METHOD FINAL metMbSerialClient
VAR_IN_OUT
	tTimeOut	: TIME;
	utQuery	    : WagoAppPlcModbus.typMbQuery;
	xTrigger	: BOOL;
	utResponse	: WagoAppPlcModbus.typMbResponse;
END_VAR
VAR_OUTPUT
	xError	: BOOL;
	uiID	: UINT;
END_VAR
VAR
	xDumyTrigger	:	BOOL;
END_VAR
IF NOT fbConfigFile.xError THEN
	(* Clear Call on Error*)
	IF fbMbClientSerial.xError THEN
		fbMbClientSerial(xConnect 	:= FALSE,
						 xTrigger 	:= xDumyTrigger,
						 utQuery  	:= utQuery,
						 utResponse := utResponse);
	END_IF;				 
    fbMbClientSerial           (xConnect    := xTrigger,
                                I_Port      := I_Port,
                                udiBaudrate := scParameter.fbudiBaudrate.udiValue,
                                usiDataBits := scParameter.fbusiDataBits.usiValue,
                                eParity     := scParameter.fbiParity.iValue,
                                eStopBits   := scParameter.fbiStopBits.iValue,
                                eHandshake  := scParameter.fbiHandshake.iValue,
                                ePhysical   := scParameter.fbiPhysikal.iValue,
                                eFrameType  := SEL(scParameter.fbxRtuOrAscii.xValue,WagoAppPlcModbus.eMbFrameType.RTU,WagoAppPlcModbus.eMbFrameType.ASCII),
                                tTimeOut    := tTimeOut,
                                utQuery     := utQuery,
                                xTrigger    := xTrigger,
                                utResponse  := utResponse,
                                xError      => xError);    
								(* Status *)
                                uiID        := fbMbClientSerial.oStatus.uiID;								
ELSE
    xError := TRUE;
END_IF;
END_METHOD

ACTION actConfig:
(* Config File *)
fbConfigFile();

scParameter.fbudiBaudrate         (_usiParaNr :=  1, ItfConfigFb := fbConfigFile , _MinInit := 9600     , _MaxInit :=  115200 );
scParameter.fbusiDataBits         (_usiParaNr :=  2, ItfConfigFb := fbConfigFile , _MinInit :=    5     , _MaxInit :=       8 );
scParameter.fbiParity             (_usiParaNr :=  3, ItfConfigFb := fbConfigFile , _MinInit :=    0     , _MaxInit :=       5 );
scParameter.fbiStopBits           (_usiParaNr :=  4, ItfConfigFb := fbConfigFile , _MinInit :=    0     , _MaxInit :=       5 );
scParameter.fbiHandshake          (_usiParaNr :=  5, ItfConfigFb := fbConfigFile , _MinInit :=    0     , _MaxInit :=       7 );
scParameter.fbiPhysikal           (_usiParaNr :=  6, ItfConfigFb := fbConfigFile , _MinInit :=    0     , _MaxInit :=       6 );
scParameter.fbxRtuOrAscii         (_usiParaNr :=  7, ItfConfigFb := fbConfigFile                                              );
END_ACTION

END_FUNCTION_BLOCK

// 30 Program Organization Units/SERVER/fbModBusServer
{warning 'Each Modbus server needs 400000 bytes of dynamic memory'}
FUNCTION_BLOCK fbModBusServer IMPLEMENTS ITF_SERVER
VAR_INPUT
    I_SerialPort                    :   WagoTypesCom.I_WagoSysComBase;
END_VAR
VAR_OUTPUT
    xError                          :   BOOL;
END_VAR
VAR
    (* Memory *)
    ayxCoil                         :   POINTER TO ARRAY[0..16#FFFF] OF BOOL;
    ayxDiscretInput                 :   POINTER TO ARRAY[0..16#FFFF] OF BOOL;  
    aywInputRegister                :   POINTER TO ARRAY[0..16#FFFF] OF WORD;
    aywHoldingRegister              :   POINTER TO ARRAY[0..16#FFFF] OF WORD; 
    xMemoryError                    :   BOOL;
    xMemoryAllocate                 :   BOOL    := TRUE;
    (* Tcp *)
    fbMbServerModelTcp              :   WagoAppPlcModbus.FbMbSlaveDataModel;
    fbMbShowAccesTcp                :   WagoAppPlcModbus.FbShowMbAccessInfo;
    fbMbTcpServer                   :   WagoAppPlcModbus.FbMbServerTcp;
    scKeepAlive                     :   WagoAppPlcModbus.typKeepAlive;
    ltLastAccesTcp                  :   LTIME;
    fbLastAccesTcp                  :   CtaAppTime.fbTimeMeasurement;
    xErrorWatchDogTcp               :   BOOL;
    xErrorTcp                       :   BOOL;
    
    (* Udp *)
    fbMbServerModelUdp              :   WagoAppPlcModbus.FbMbSlaveDataModel;
    fbMbShowAccesUdp                :   WagoAppPlcModbus.FbShowMbAccessInfo;
    fbMbUdpServer                   :   WagoAppPlcModbus.fbMbServerUdp;
    ltLastAccesUdp                  :   LTIME;
    fbLastAccesUdp                  :   CtaAppTime.fbTimeMeasurement;  
    xErrorWatchDogUdp               :   BOOL;  
    xErrorUdp                       :   BOOL;
    
    (* Serial *)
    fbMbServerModelSerial           :   WagoAppPlcModbus.FbMbSlaveDataModel;
    fbMbShowAccesSerial             :   WagoAppPlcModbus.FbShowMbAccessInfo;
    fbMbRtuSerialServer             :   WagoAppPlcModbus.FbMbServerSerial;
    ltLastAccesSerial               :   LTIME;
    fbLastAccesSerial               :   CtaAppTime.fbTimeMeasurement;
    xErrorWatchDogSerial            :   BOOL;    
    xErrorSerial                    :   BOOL;
    
    (* Parameter *)
    fbConfigFile                    :   CtaSysConfig.fbConfigFile;
    scParameter                     :   scModBusServerParameter;
END_VAR

actConfig();
IF xMemoryAllocate AND NOT xMemoryError THEN
    ayxCoil             := __NEW(BOOL,16#10000);
    ayxDiscretInput     := __NEW(BOOL,16#10000);
    aywInputRegister    := __NEW(WORD,16#10000);
    aywHoldingRegister  := __NEW(WORD,16#10000);
    IF ayxCoil <> 0 AND ayxDiscretInput <> 0 AND aywInputRegister <> 0 AND aywHoldingRegister <> 0 THEN
        xMemoryAllocate     := FALSE;     
    ELSE 
        xMemoryError := TRUE;   
    END_IF;
END_IF;
IF  NOT xMemoryAllocate AND NOT xMemoryError THEN
    IF SIZEOF(ayxCoil^) = 65536 AND SIZEOF(ayxDiscretInput^) = 65536 AND SIZEOF(aywInputRegister^) = 131072 AND SIZEOF(aywHoldingRegister^) = 131072 THEN
        IF NOT fbConfigFile.xError THEN
            actModBusServerSerial();
            actModBusServerTcp();
            actModBusServerUdp();
        END_IF;    
        xMemoryError := FALSE;
    ELSE
        xMemoryError := TRUE;    
    END_IF
END_IF;
(* Error *)
xError := fbConfigFile.xError OR xErrorTcp OR xErrorUdp OR xErrorSerial OR xMemoryError;

ACTION actConfig:
(* Config File *)
fbConfigFile();

scParameter.scSerial.fbbyUnitId            (_usiParaNr :=  1, ItfConfigFb := fbConfigFile , _MinInit :=    0     , _MaxInit :=     247 ); 
scParameter.scSerial.fbxEnable             (_usiParaNr :=  2, ItfConfigFb := fbConfigFile                                              );
scParameter.scSerial.fbudiBaudrate         (_usiParaNr :=  3, ItfConfigFb := fbConfigFile , _MinInit := 9600     , _MaxInit :=   19600 );
scParameter.scSerial.fbusiDataBits         (_usiParaNr :=  4, ItfConfigFb := fbConfigFile , _MinInit :=    5     , _MaxInit :=       8 );
scParameter.scSerial.fbiParity             (_usiParaNr :=  5, ItfConfigFb := fbConfigFile , _MinInit :=    0     , _MaxInit :=       5 );
scParameter.scSerial.fbiStopBits           (_usiParaNr :=  6, ItfConfigFb := fbConfigFile , _MinInit :=    0     , _MaxInit :=       5 );
scParameter.scSerial.fbiHandshake          (_usiParaNr :=  7, ItfConfigFb := fbConfigFile , _MinInit :=    0     , _MaxInit :=       7 );
scParameter.scSerial.fbiPhysikal           (_usiParaNr :=  8, ItfConfigFb := fbConfigFile , _MinInit :=    0     , _MaxInit :=       6 );
scParameter.scSerial.fbxRtuOrAscii         (_usiParaNr :=  9, ItfConfigFb := fbConfigFile                                              );
scParameter.scSerial.fbxEnableWatchDog     (_usiParaNr := 10, ItfConfigFb := fbConfigFile                                              );
scParameter.scSerial.fbtWatchDog           (_usiParaNr := 11, ItfConfigFb := fbConfigFile , _MinInit := T#1S     , _MaxInit :=   T#10M );
scParameter.scTcp.fbxEnable                (_usiParaNr := 12, ItfConfigFb := fbConfigFile                                              );
scParameter.scTcp.fbbyUnitId               (_usiParaNr := 13, ItfConfigFb := fbConfigFile , _MinInit :=    0     , _MaxInit :=     255 ); 
scParameter.scTcp.fbwPort                  (_usiParaNr := 14, ItfConfigFb := fbConfigFile , _MinInit :=    0     , _MaxInit := 16#FFFF );
scParameter.scTcp.fbxKeepAlive             (_usiParaNr := 15, ItfConfigFb := fbConfigFile                                              );
scParameter.scTcp.fbtMaxIdleTime           (_usiParaNr := 16, ItfConfigFb := fbConfigFile , _MinInit := T#1S     , _MaxInit :=   T#10M );
scParameter.scTcp.fbtIntervall             (_usiParaNr := 17, ItfConfigFb := fbConfigFile , _MinInit := T#1S     , _MaxInit :=   T#10M );
scParameter.scTcp.fbudiProbes              (_usiParaNr := 18, ItfConfigFb := fbConfigFile , _MinInit :=    0     , _MaxInit :=     500 );
scParameter.scTcp.fbxEnableWatchDog        (_usiParaNr := 19, ItfConfigFb := fbConfigFile                                              );
scParameter.scTcp.fbtWatchDog              (_usiParaNr := 20, ItfConfigFb := fbConfigFile , _MinInit := T#50MS   , _MaxInit :=   T#10M );
scParameter.scUdp.fbxEnable                (_usiParaNr := 21, ItfConfigFb := fbConfigFile                                              );
scParameter.scUdp.fbbyUnitId               (_usiParaNr := 22, ItfConfigFb := fbConfigFile , _MinInit :=    0     , _MaxInit :=     255 ); 
scParameter.scUdp.fbwPort                  (_usiParaNr := 23, ItfConfigFb := fbConfigFile , _MinInit :=    0     , _MaxInit := 16#FFFF );
scParameter.scUdp.fbxEnableWatchDog        (_usiParaNr := 24, ItfConfigFb := fbConfigFile                                              );
scParameter.scUdp.fbtWatchDog              (_usiParaNr := 25, ItfConfigFb := fbConfigFile , _MinInit := T#1S     , _MaxInit :=   T#10M );
END_ACTION

ACTION actModBusServerTcp:
(* Server Memory Tcp*)
fbMbServerModelTcp(     bUnitId             := scParameter.scTcp.fbbyUnitId.byValue,
                        IIdentifyObject     := GVL_CtaModBus.fbDeviceName,
                        axDiscreteInputs    := ayxDiscretInput^,
                        axCoils             := ayxCoil^,
                        awInputRegisters    := aywInputRegister^,
                        awHoldingRegisters  := aywHoldingRegister^); 
                        
(* Tcp Server *)
IF scParameter.scTcp.fbxEnable.xValue THEN
    scKeepAlive.xEnable                     := scParameter.scTcp.fbxKeepAlive.xValue;
    scKeepAlive.tMaxIdleTime                := scParameter.scTcp.fbtMaxIdleTime.tValue;
    scKeepAlive.tInterval                   := scParameter.scTcp.fbtIntervall.tValue;
    scKeepAlive.udiProbes                   := scParameter.scTcp.fbudiProbes.udiValue;
    fbMbTcpServer(      xOpen               := scParameter.scTcp.fbxEnable.xValue,
                        wPort               := scParameter.scTcp.fbwPort.wValue,
                        utKeepAlive         := scKeepAlive,
                        eFrameType          := WagoAppPlcModbus.eMbFrameType.ETHERNET,
                        I_MbDataModel       := fbMbServerModelTcp.I_MbDataModel);
ELSIF fbMbTcpServer.xOpen THEN
    fbMbTcpServer(      xOpen               := FALSE,
                        I_MbDataModel       := fbMbServerModelTcp.I_MbDataModel);                           
END_IF;                        

(* Acces Info *)
fbMbShowAccesTcp    (   oMbAccessInfo := fbMbServerModelTcp.oMbAccessInfo);   

(* Acces Time *)
IF fbMbServerModelTcp.isReadAccess OR fbMbServerModelTcp.isWriteAccess THEN
    fbLastAccesTcp.Start();
    ltLastAccesTcp := fbLastAccesTcp.Stop();
ELSE
    ltLastAccesTcp := fbLastAccesTcp.Stop();
END_IF;

(* WatchDog *)
IF scParameter.scTcp.fbxEnableWatchDog.xValue THEN
    xErrorWatchDogTcp := TO_LTIME(scParameter.scTcp.fbtWatchDog.tValue) < ltLastAccesTcp;
ELSE
    xErrorWatchDogTcp := FALSE;
END_IF;

(* Error *)
xErrorTcp := fbConfigFile.xError OR fbMbServerModelTcp.xError OR fbMbTcpServer.xError OR xErrorWatchDogTcp;
END_ACTION

ACTION actModBusServerUdp:
(* Server Memory Udp*)
fbMbServerModelUdp(     bUnitId             := scParameter.scUdp.fbbyUnitId.byValue,
                        IIdentifyObject     := GVL_CtaModBus.fbDeviceName,
                        axDiscreteInputs    := ayxDiscretInput^,
                        axCoils             := ayxCoil^,
                        awInputRegisters    := aywInputRegister^,
                        awHoldingRegisters  := aywHoldingRegister^);  
                        
(* UDP Server *)
IF scParameter.scUdp.fbxEnable.xValue THEN
    fbMbUdpServer(      xOpen               := scParameter.scUdp.fbxEnable.xValue,
                        wPort               := scParameter.scUdp.fbwPort.wValue,
                        eFrameType          := WagoAppPlcModbus.eMbFrameType.ETHERNET,
                        I_MbDataModel       := fbMbServerModelUdp.I_MbDataModel);
ELSIF fbMbUdpServer.xOpen THEN
    fbMbUdpServer(      xOpen               := FALSE,
                        I_MbDataModel       := fbMbServerModelUdp.I_MbDataModel);                        
END_IF;                          

(* Acces Info *)
fbMbShowAccesUdp    (   oMbAccessInfo := fbMbServerModelUdp.oMbAccessInfo); 

(* Acces Time *)
IF fbMbServerModelUdp.isReadAccess OR fbMbServerModelUdp.isWriteAccess THEN
    fbLastAccesUdp.Start();
    ltLastAccesUdp := fbLastAccesSerial.Stop();
ELSE
    ltLastAccesUdp := fbLastAccesSerial.Stop();
END_IF;

(* WatchDog *)
IF scParameter.scUdp.fbxEnableWatchDog.xValue THEN
    xErrorWatchDogUdp := TO_LTIME(scParameter.scUdp.fbtWatchDog.tValue) < ltLastAccesUdp;
ELSE
    xErrorWatchDogUdp := FALSE;
END_IF;

(* Error *)
xErrorUdp := fbConfigFile.xError OR fbMbServerModelUdp.xError OR fbMbUdpServer.xError OR xErrorWatchDogUdp;
END_ACTION

ACTION actModBusServerSerial:
(* Server Memory Serial*)
fbMbServerModelSerial(  bUnitId             := scParameter.scSerial.fbbyUnitId.byValue,
                        IIdentifyObject     := GVL_CtaModBus.fbDeviceName,
                        axDiscreteInputs    := ayxDiscretInput^,
                        axCoils             := ayxCoil^,
                        awInputRegisters    := aywInputRegister^,
                        awHoldingRegisters  := aywHoldingRegister^);  
                        
(* SERIAL Server *)           
IF scParameter.scSerial.fbxEnable.xValue THEN    
	IF __QUERYINTERFACE(I_SerialPort,I_SerialPort) THEN
		(* Server Run*) 
		fbMbRtuSerialServer(xConnect            := scParameter.scSerial.fbxEnable.xValue,
							I_Port              := I_SerialPort,
							udiBaudrate         := scParameter.scSerial.fbudiBaudrate.udiValue,
							usiDataBits         := scParameter.scSerial.fbusiDataBits.usiValue,
							eParity             := scParameter.scSerial.fbiParity.iValue,
							eStopBits           := scParameter.scSerial.fbiStopBits.iValue,
							eHandshake          := scParameter.scSerial.fbiHandshake.iValue,
							ePhysical           := scParameter.scSerial.fbiPhysikal.iValue,
							eFrameType          := SEL(scParameter.scSerial.fbxRtuOrAscii.xValue,WagoAppPlcModbus.eMbFrameType.RTU,WagoAppPlcModbus.eMbFrameType.ASCII),
							I_MbDataModel       := fbMbServerModelSerial.I_MbDataModel);
   	END_IF;                     
    (* Acces Info *)
    fbMbShowAccesSerial (   oMbAccessInfo := fbMbServerModelSerial.oMbAccessInfo); 
    
    (* Acces Time *)
    IF fbMbServerModelSerial.isReadAccess OR fbMbServerModelSerial.isWriteAccess THEN
        fbLastAccesSerial.Start();
        ltLastAccesSerial := fbLastAccesSerial.Stop();
    ELSE
        ltLastAccesSerial := fbLastAccesSerial.Stop();
    END_IF;
    
    (* WatchDog *)
    IF scParameter.scSerial.fbxEnableWatchDog.xValue THEN
        xErrorWatchDogSerial := TO_LTIME(scParameter.scSerial.fbtWatchDog.tValue) < ltLastAccesSerial;
    ELSE
        xErrorWatchDogSerial := FALSE;
    END_IF;                        
                        
ELSIF fbMbRtuSerialServer.xConnect THEN
    (* Server Disconnect *)
    fbMbRtuSerialServer(xConnect            := FALSE,
                        I_Port              := I_SerialPort,
                        I_MbDataModel       := fbMbServerModelSerial.I_MbDataModel);   
ELSE
    xErrorWatchDogSerial := FALSE;
    ltLastAccesSerial    := fbLastAccesSerial.Stop();
END_IF;                        



(* Error *)
xErrorSerial := fbConfigFile.xError OR fbMbServerModelSerial.xError OR fbMbRtuSerialServer.xError OR xErrorWatchDogSerial;
END_ACTION

METHOD metGetCoil : BOOL
VAR_INPUT
    wAdr          : WORD;
END_VAR
IF NOT xMemoryAllocate AND NOT xMemoryError THEN
	IF wAdr >= LOWER_BOUND(ayxCoil^,1) AND wAdr <= UPPER_BOUND(ayxCoil^,1) THEN
    	metGetCoil := ayxCoil^[wAdr];
	END_IF;
END_IF;
END_METHOD

METHOD metSetDiscretInput : BOOL
VAR_INPUT
    wAdr          : WORD;
    xValue        : BOOL;
END_VAR
IF NOT xMemoryAllocate AND NOT xMemoryError THEN
	IF wAdr >= LOWER_BOUND(ayxDiscretInput^,1) AND wAdr <= UPPER_BOUND(ayxDiscretInput^,1) THEN
    	ayxDiscretInput^[wAdr] := xValue;
	END_IF;
END_IF;
END_METHOD

METHOD metGetHoldingRegister : WORD
VAR_INPUT
    wAdr          : WORD;
END_VAR
IF NOT xMemoryAllocate AND NOT xMemoryError THEN
	IF wAdr >= LOWER_BOUND(aywHoldingRegister^,1) AND wAdr <= UPPER_BOUND(aywHoldingRegister^,1) THEN
    	metGetHoldingRegister := aywHoldingRegister^[wAdr];
	END_IF;
END_IF;
END_METHOD

METHOD metSetInputRegister : BOOL
VAR_INPUT
    wAdr          : WORD;
    wValue        : WORD;
END_VAR
IF NOT xMemoryAllocate AND NOT xMemoryError THEN
	IF wAdr >= LOWER_BOUND(aywInputRegister^,1) AND wAdr <= UPPER_BOUND(aywInputRegister^,1) THEN
    	aywInputRegister^[wAdr] := wValue;
	END_IF;
END_IF;
END_METHOD

METHOD metAddSerialControll : BOOL
VAR_INPUT
    I_DataAccesListener :   WagoAppPlcModbus.I_DataAccessListener;
END_VAR
fbMbServerModelSerial.RegisterDataAccessListener(I_DataAccesListener);
END_METHOD

METHOD metAddTcpControll : BOOL
VAR_INPUT
    I_DataAccesListener :   WagoAppPlcModbus.I_DataAccessListener;
END_VAR
fbMbServerModelTcp.RegisterDataAccessListener(I_DataAccesListener);
END_METHOD

METHOD metAddUdpControll : BOOL
VAR_INPUT
    I_DataAccesListener :   WagoAppPlcModbus.I_DataAccessListener;
END_VAR
fbMbServerModelUdp.RegisterDataAccessListener(I_DataAccesListener);
END_METHOD

METHOD metSetHoldingRegister : BOOL
VAR_INPUT
    wAdr          : WORD;
    wValue        : WORD;
END_VAR
IF NOT xMemoryAllocate AND NOT xMemoryError THEN
	IF wAdr >= LOWER_BOUND(aywHoldingRegister^,1) AND wAdr <= UPPER_BOUND(aywHoldingRegister^,1) THEN
    	aywHoldingRegister^[wAdr] := wValue;
	END_IF;
END_IF;
END_METHOD

METHOD metSetCoil : BOOL
VAR_INPUT
    wAdr          : WORD;
    xValue        : BOOL;
END_VAR
IF NOT xMemoryAllocate AND NOT xMemoryError THEN
	IF wAdr >= LOWER_BOUND(ayxCoil^,1) AND wAdr <= UPPER_BOUND(ayxCoil^,1) THEN
    	ayxCoil^[wAdr] := xValue;
	END_IF;
END_IF;
END_METHOD

END_FUNCTION_BLOCK

// 21 Interface/SERVER/ITF_SERVER
INTERFACE ITF_SERVER EXTENDS CtaAppModbus.ITF_SERVER

METHOD metAddSerialControll : BOOL
VAR_INPUT
    I_DataAccesListener :   WagoAppPlcModbus.I_DataAccessListener;
END_VAR
END_METHOD

METHOD metAddTcpControll : BOOL
VAR_INPUT
    I_DataAccesListener :   WagoAppPlcModbus.I_DataAccessListener;
END_VAR
END_METHOD

METHOD metAddUdpControll : BOOL
VAR_INPUT
    I_DataAccesListener :   WagoAppPlcModbus.I_DataAccessListener;
END_VAR
END_METHOD

END_INTERFACE

// 30 Program Organization Units/CLIENT/NETWORK Client/TCP/fbMbTcpClient
FUNCTION_BLOCK fbMbTcpClient EXTENDS CtaSysBase.fbBASE IMPLEMENTS ITF_MbClient ,ITF_TCP_NODE                 
VAR_INPUT
    ITF_MbPortControll          : ITF_MbPortControllTcp;   
END_VAR
VAR_OUTPUT                      
    xError                      : BOOL;
END_VAR
VAR    
    (* Tcp Client *)
	ITF_BMK 					: CtaAppBmk.ITF_BMK;			
    xComAktive                  : BOOL;
    xDisabled                   : BOOL;
    xAllJobsDone                : BOOL;
    bIdOfCall                   : BYTE;
    byUnitId                    : BYTE;
    ITF_MbPortControllQuerry    : ITF_MbPortControllTcp;
    xPortControllError          : BOOL;
    scKeepAlive                 : WagoAppPlcModbus.typKeepAlive;
    xErrorMbClientTcp           : BOOL;
    uiIdMbClientTcp             : UINT;

    (* Main State *)
    uiCountErrors               : UINT;   
    usiState                    : USINT := 1;
    fbTIMEFcs                   : CtaAppTime.fbTimeMeasurement;
    ltMessungFcs                : LTIME; 
    
    (* Scan Rate *)
    TON_ScanRate                : TON;
    tonDelayRead				: Standard.TON;
	tonDelayWrite				: Standard.TON;
	xTrigDelayRead				: BOOL;
	xTrigDelayWrite				: BOOL;        
    (* FC1 *)
    fbJobFc1                    : fbJOB;
    xTrigFc1                    : BOOL;
    fbTIMEFc1                   : CtaAppTime.fbTimeMeasurement;
    ltMessungFc1                : LTIME;   
    (* FC2 *)
    fbJobFc2                    : fbJOB;
    xTrigFc2                    : BOOL; 
    fbTIMEFc2                   : CtaAppTime.fbTimeMeasurement;
    ltMessungFc2                : LTIME;    
    (* FC3 *)
    fbJobFc3                    : fbJOB;
    xTrigFc3                    : BOOL;      
    fbTIMEFc3                   : CtaAppTime.fbTimeMeasurement;
    ltMessungFc3                : LTIME;         
    (* FC4 *)
    fbJobFc4                    : fbJOB;
    xTrigFc4                    : BOOL;      
    fbTIMEFc4                   : CtaAppTime.fbTimeMeasurement;
    ltMessungFc4                : LTIME;  
    (* FC5 *)
    fbJobFc5                    : fbJOB;
    xTrigFc5                    : BOOL;      
    fbTIMEFc5                   : CtaAppTime.fbTimeMeasurement;
    ltMessungFc5                : LTIME;    
    (* FC6 *)
    fbJobFc6                    : fbJOB;
    xTrigFc6                    : BOOL;      
    fbTIMEFc6                   : CtaAppTime.fbTimeMeasurement;
    ltMessungFc6                : LTIME;       
    (* FC15 *)
    fbJobFc15                   : fbJOB;
    xTrigFc15                   : BOOL;   
    fbTIMEFc15                  : CtaAppTime.fbTimeMeasurement;
    ltMessungFc15               : LTIME;    
    (* FC16 *)   
    fbJobFc16                   : fbJOB;             
    xTrigFc16                   : BOOL;
    fbTIMEFc16                  : CtaAppTime.fbTimeMeasurement;
    ltMessungFc16               : LTIME;      
(* FC43 *)   
    fbIdentifyObject			: WagoAppPlcModbus.FbIdentifyBaseObject;
	fbIdentifyMember3			: WagoAppPlcModbus.FbIdentifyMember_STRING(fbIdentifyObject,3);
	fbIdentifyMember4			: WagoAppPlcModbus.FbIdentifyMember_STRING(fbIdentifyObject,4);
	utIdentifyQuerry			: WagoAppPlcModbus.typMbQuery;
	utIdentifyResponse			: WagoAppPlcModbus.typMbResponse;           
    xTrigFc43                   : BOOL;
	xActiveFc43					: BOOL;
	xDoneFc43					: BOOL;
	tTimeOutFc43				: TIME;
    fbTIMEFc43                  : CtaAppTime.fbTimeMeasurement;
    ltMessungFc43               : LTIME;	
    (* Parameter *)
    fbConfigFile                : CtaSysConfig.fbConfigFile;
    scParameter                 : scTcpClientParameter;
END_VAR

(* Config *)
actConfig();
(* Unit ID *)
byUnitId := scParameter.fbbyUnitId.byValue;
(* Is Enabled *)
IF scParameter.fbxEnable.xValue AND byUnitId <> 0 THEN
    (* Port Sync *)
    IF __QUERYINTERFACE(ITF_MbPortControll,ITF_MbPortControllQuerry) THEN
        xPortControllError := FALSE;  
        IF ITF_MbPortControllQuerry.metSyncClient(xAllJobsDone,bIdOfCall,THIS^) THEN    
			(* Delay *)
			actDelay();
            (* Keep Alive *)
            actKeepAlive();
            (* FC1 *)
            actFC01();
            (* FC2 *)
            actFC02();
            (* FC3 *)
            actFC03();
            (* FC4 *)
            actFC04();
            (* FC5 *)
            actFC05();
            (* FC6 *)
            actFC06();			
            (* FC15 *)
            actFC15();
            (* FC16 *)
            actFC16(); 
			(* FC43 *)
			actFC43();
        END_IF;
    ELSE
        xPortControllError := TRUE;    
    END_IF;    
    IF usiState >= 10 OR usiState = 0 THEN
        (* Check if all Jobs Done *)
        IF  fbJobFc1.xAllJobsDone  AND
            fbJobFc2.xAllJobsDone  AND
            fbJobFc3.xAllJobsDone  AND
            fbJobFc4.xAllJobsDone  AND
            fbJobFc5.xAllJobsDone  AND
            fbJobFc6.xAllJobsDone  AND			
            fbJobFc15.xAllJobsDone AND
            fbJobFc16.xAllJobsDone THEN
            (*Scan Rate *)
            TON_ScanRate(IN := NOT TON_ScanRate.Q,
                         PT := scParameter.fbtScanRate.tValue);
            xAllJobsDone := TRUE;             
            IF TON_ScanRate.Q THEN
                fbJobFc1.proAllJobsDone  := FALSE;
                fbJobFc2.proAllJobsDone  := FALSE;   
                fbJobFc3.proAllJobsDone  := FALSE;  
                fbJobFc4.proAllJobsDone  := FALSE;   
                fbJobFc5.proAllJobsDone  := FALSE;  
                fbJobFc6.proAllJobsDone  := FALSE; 	
                fbJobFc15.proAllJobsDone := FALSE;  
                fbJobFc16.proAllJobsDone := FALSE; 
				xAllJobsDone             := FALSE;       
                usiState := 1;
                (* Timer stopp *) 
                ltMessungFcs := fbTIMEFcs.stop();             
                (* Timer start *) 
                fbTIMEFcs.Start();      
            END_IF;        
        ELSE    
            usiState := 1;
        END_IF;   
    END_IF;

    xComAktive := fbJobFc1.wCountJobs  <> 0 OR 
                  fbJobFc2.wCountJobs  <> 0 OR
                  fbJobFc3.wCountJobs  <> 0 OR 
                  fbJobFc4.wCountJobs  <> 0 OR 
                  fbJobFc15.wCountJobs <> 0 OR
                  fbJobFc16.wCountJobs <> 0 ;  
                      
    (* Get Errors *)
    xError :=  fbJobFc1.eError <> WagoAppPlcModbus.eErrorModbus.OK OR 
               fbJobFc2.eError <> WagoAppPlcModbus.eErrorModbus.OK OR 
               fbJobFc3.eError <> WagoAppPlcModbus.eErrorModbus.OK OR 
               fbJobFc4.eError <> WagoAppPlcModbus.eErrorModbus.OK OR 
			   fbJobFc5.eError <> WagoAppPlcModbus.eErrorModbus.OK OR
			   fbJobFc6.eError <> WagoAppPlcModbus.eErrorModbus.OK OR
              fbJobFc15.eError <> WagoAppPlcModbus.eErrorModbus.OK OR 
              fbJobFc16.eError <> WagoAppPlcModbus.eErrorModbus.OK OR 
              fbConfigFile.xError                                  OR
              xPortControllError; 
    IF NOT xError THEN
       uiCountErrors := 0;
    END_IF;    
ELSE
    (* Reset States *)
    (* Port Sync *)
    IF __QUERYINTERFACE(ITF_MbPortControll,ITF_MbPortControllQuerry) THEN
        xPortControllError := FALSE;  
        xAllJobsDone       := FALSE;
        usiState           := 0;
        xError             := FALSE;
        xComAktive         := FALSE;
        xDisabled          := TRUE;
        ITF_MbPortControllQuerry.metSyncClient(xDisabled,bIdOfCall,THIS^);
    END_IF;      
END_IF;

ACTION actKeepAlive:
scKeepAlive.xEnable                     := scParameter.fbxKeepAlive.xValue;
scKeepAlive.tMaxIdleTime                := scParameter.fbtMaxIdleTime.tValue;
scKeepAlive.tInterval                   := scParameter.fbtIntervall.tValue;
scKeepAlive.udiProbes                   := scParameter.fbudiProbes.udiValue;
END_ACTION

//FB_Init ist immer implizit verfügbar und wird primär für die Initialisierung verwendet.
//Der Rückgabewert wird nicht ausgewertet. Für gezielte Einflussnahme können Sie
//die Methoden explizit deklarieren und darin mit dem Standard-Initialisierungscode 
//zusätzlichen Code bereitstellen. Sie können den Rückgabewert auswerten.
METHOD FB_Init: BOOL
VAR_INPUT    
bInitRetains: BOOL; // TRUE: Die Retain-Variablen werden initialisiert (Reset warm / Reset kalt)    
bInCopyCode: BOOL;  // TRUE: Die Instanz wird danach in den Kopiercode kopiert (Online-Change)
END_VAR
xTrigFc1    := FALSE;
xTrigFc2    := FALSE;
xTrigFc3    := FALSE;
xTrigFc4    := FALSE;
xTrigFc15   := FALSE;
xTrigFc16   := FALSE;
usiState    := 0;
END_METHOD

METHOD PRIVATE FINAL metCheckOnError : BOOL
VAR_INPUT
    xError  :  BOOL;
END_VAR
IF xError THEN
    uiCountErrors  := uiCountErrors + 1;
    metCheckOnError := TRUE;
END_IF
END_METHOD

METHOD FINAL metFc4ReadInputRegister
VAR_INPUT
    wADR                :   WORD;
    pWord               :   POINTER TO WORD;
    uiQuantity          :   UINT;               // Anzahl Words Max 123
    wOffset             :   WORD;               // Pointer Offset wenn WORD Array > 123   
END_VAR
VAR
    diCurrentJop        :   DINT;
    uiFor               :   UINT;
    pBaseAdr            :   POINTER TO WORD;
END_VAR
(* Limit Read Input Register *)
uiQuantity := LIMIT(1,uiQuantity,123);
(* Check if valid Pointer and Adress *)
IF pWord <> 0 AND wOffset + uiQuantity <= 16#FFFF + 1 AND wADR <= 16#FFFF THEN
    (* Link Adress *)
    fbJobFc4.bUnitId       := byUnitId;   
    fbJobFc4.bFunctionCode := 4;
    fbJobFc4.xIsBoolQuerry := FALSE;
    fbJobFc4.xIsSerialJob  := FALSE;     
    fbJobFc4.metCheckQuerryAdr(wADR,uiQuantity,pWord,wOffset);        
END_IF;
END_METHOD

ACTION actFC04:
(* Trig FC4 *)
IF fbJobFc4.xIsLinked AND fbJobFc4.xIsQuerryReady AND NOT fbJobFc4.xIsLocked AND NOT fbJobFc4.xAllJobsDone AND tonDelayRead.Q THEN
    fbJobFc4.metLock();
    xTrigFc4       := TRUE;
    fbTIMEFc4.Start();
ELSIF usiState = 4 AND (NOT fbJobFc4.xIsLinked OR fbJobFc4.xAllJobsDone) THEN
    usiState                := usiState + 1;    
    fbJobFc4.proAllJobsDone := TRUE;
END_IF

(* Send Querry *)
IF usiState = 4 AND xTrigFc4 THEN
	xTrigDelayRead 	:= FALSE;
    ITF_MbPortControllQuerry.metMbTcpClient(    stIp        := scParameter.fbstIp.stValue,
                                                wPort       := scParameter.fbwPort.wValue,
                                                scKeepAlive := scKeepAlive,
                                                tTimeOut    := scParameter.fbtTimeOut.tValue,
                                                utQuery     := fbJobFc4.utQuery,
                                                xTrigger    := xTrigFc4,
                                                utResponse  := fbJobFc4.utResponse,
                                                xError      => xErrorMbClientTcp,
                                                uiID        => uiIdMbClientTcp);       
END_IF;
(* Get Response *) 
IF usiState = 4 AND NOT xTrigFc4 AND fbJobFc4.xIsLocked AND NOT fbJobFc4.xJobDone THEN
    usiState            := usiState + 1;
    ltMessungFc4        := fbTIMEFc4.Stop();
    metCheckOnError(xErrorMbClientTcp);
    fbJobFc4.metCallAfterResponse(xErrorMbClientTcp,uiIdMbClientTcp);
END_IF;
END_ACTION

METHOD FINAL metFc2ReadDiscretInput
VAR_INPUT
    wADR                :   WORD;
    pByte               :   POINTER TO BYTE;
    uiQuantity          :   UINT;               // Anzahl BOOL Max 1968
    wOffset             :   WORD;               // Pointer Offset wenn BOOL Array > 1968    
END_VAR
VAR
    diCurrentJop        :   DINT;
    uiFor               :   UINT;
    usiCountWords       :   UINT;    
    wTempValue          :   WORD;
    pBaseAdr            :   POINTER TO BYTE;
END_VAR
(* Limit Discret Inputs *)
uiQuantity := LIMIT(1,uiQuantity,1968);
(* Check if valid Pointer and Adress *)
IF pByte <> 0 AND wOffset + uiQuantity <= 16#FFFF + 1 AND wADR <= 16#FFFF THEN
    (* Link Adress *)
    fbJobFc2.bUnitId       := byUnitId;
    fbJobFc2.bFunctionCode := 2;
    fbJobFc2.xIsBoolQuerry := TRUE;
    fbJobFc2.xIsSerialJob  := FALSE;    
    fbJobFc2.metCheckQuerryAdr(wADR,uiQuantity,pByte,wOffset);    
END_IF;
END_METHOD

ACTION actFC15:
(* Trig FC15 *)
IF fbJobFc15.xIsLinked AND fbJobFc15.xIsQuerryReady AND NOT fbJobFc15.xIsLocked AND NOT fbJobFc15.xAllJobsDone AND tonDelayWrite.Q THEN
    fbJobFc15.metLock();
    xTrigFc15       := TRUE;
    fbTIMEFc15.Start();
ELSIF usiState = 7 AND (NOT fbJobFc15.xIsLinked OR fbJobFc15.xAllJobsDone) THEN
    usiState                    := usiState + 1;  
    fbJobFc15.proAllJobsDone    := TRUE;  
END_IF;

(* Send Querry *)
IF usiState = 7 AND xTrigFc15 THEN
	xTrigDelayWrite := FALSE;
    ITF_MbPortControllQuerry.metMbTcpClient(    stIp        := scParameter.fbstIp.stValue,
                                                wPort       := scParameter.fbwPort.wValue,
                                                scKeepAlive := scKeepAlive,
                                                tTimeOut    := scParameter.fbtTimeOut.tValue,
                                                utQuery     := fbJobFc15.utQuery,
                                                xTrigger    := xTrigFc15,
                                                utResponse  := fbJobFc15.utResponse,
                                                xError      => xErrorMbClientTcp,
                                                uiID        => uiIdMbClientTcp);       
END_IF;
(* Get Response *) 
IF usiState = 7 AND NOT xTrigFc15 AND fbJobFc15.xIsLocked AND NOT fbJobFc15.xJobDone THEN
    usiState             := usiState + 1;
    ltMessungFc15        := fbTIMEFc15.Stop();
    metCheckOnError(xErrorMbClientTcp);
    fbJobFc15.metCallAfterResponse(xErrorMbClientTcp,uiIdMbClientTcp);
END_IF;
END_ACTION

METHOD FINAL metFc1ReadCoils
VAR_INPUT
    wADR                :   WORD;
    pByte               :   POINTER TO BYTE;
    uiQuantity          :   UINT;               // Anzahl Coils Max 1968
    wOffset             :   WORD;               // Pointer Offset wenn BOOL Array > 1968     
END_VAR
VAR
    diCurrentJop        :   DINT;
    uiFor               :   UINT;
    usiCountWords       :   UINT;
    wTempValue          :   WORD;
END_VAR
(* Limit Coils *)
uiQuantity := LIMIT(1,uiQuantity,1968);
(* Check if valid Pointer and Adress *)
IF pByte <> 0 AND wOffset + uiQuantity <= 16#FFFF + 1 AND wADR <= 16#FFFF THEN
    (* Link Adress *)
    fbJobFc1.bUnitId       := byUnitId;
    fbJobFc1.bFunctionCode := 1;
    fbJobFc1.xIsBoolQuerry := TRUE;
    fbJobFc1.xIsSerialJob  := FALSE;    
    fbJobFc1.metCheckQuerryAdr(wADR,uiQuantity,pByte,wOffset);        
END_IF;
END_METHOD

METHOD FINAL metFc3ReadHoldingRegister
VAR_INPUT
    wADR                :   WORD;
    pWord               :   POINTER TO WORD;
    uiQuantity          :   UINT;               // Anzahl Words Max 123
    wOffset             :   WORD;               // Pointer Offset wenn WORD Array > 123    
END_VAR
VAR
    diCurrentJop        :   DINT;
    uiFor               :   UINT;
    pBaseAdr            :   POINTER TO WORD;
END_VAR
(* Limit Holding Register *)
uiQuantity := LIMIT(1,uiQuantity,123);
(* Check if valid Pointer and Adress *)
IF pWord <> 0 AND wOffset + uiQuantity <= 16#FFFF + 1 AND wADR <= 16#FFFF THEN
    (* Link Adress *)
    fbJobFc3.bUnitId       := byUnitId;
    fbJobFc3.bFunctionCode := 3;
    fbJobFc3.xIsBoolQuerry := FALSE;
    fbJobFc3.xIsSerialJob  := FALSE;       
    fbJobFc3.metCheckQuerryAdr(wADR,uiQuantity,pWord,wOffset);     
END_IF;
END_METHOD

METHOD FINAL metFc15WriteMultipleCoil
VAR_INPUT
    wADR                :   WORD;
    pByte               :   POINTER TO BYTE;
    uiQuantity          :   UINT;               // Anzahl Coils Max 1968   
    wOffset             :   WORD;               // Pointer Offset wenn BOOL Array > 1968     
END_VAR
VAR
    diCurrentJop        :   DINT;
    uiFor               :   UINT;
    usiCountWords       :   UINT;
    wTempValue          :   WORD;    
END_VAR
(* Limit Write Multiple Coil *)
uiQuantity := LIMIT(1,uiQuantity,1968);
(* Check if valid Pointer and Adress *)
IF pByte <> 0 AND wOffset + uiQuantity <= 16#FFFF + 1 AND wADR <= 16#FFFF THEN
    (* Link Adress *)
    fbJobFc15.bUnitId       := byUnitId;
    fbJobFc15.bFunctionCode := 15;
    fbJobFc15.xIsBoolQuerry := TRUE;
    fbJobFc15.xIsSerialJob  := FALSE;        
    fbJobFc15.metCheckQuerryAdr(wADR,uiQuantity,pByte,wOffset);    
END_IF;
END_METHOD

METHOD FINAL metFc16WriteHoldingRegisters
VAR_INPUT
    wADR                :   WORD;
    pWord               :   POINTER TO WORD;
    uiQuantity          :   UINT;               // Anzahl Words Max 123
    wOffset             :   WORD;               // Pointer Offset wenn Array > 123 WORD    
END_VAR
VAR
    diCurrentJop        :   DINT;
    uiFor               :   UINT;
END_VAR
(* Limit Write Holding Registers *)
uiQuantity := LIMIT(1,uiQuantity,123);
(* Check if valid Pointer and Adress *)
IF pWord <> 0 AND wOffset + uiQuantity <= 16#FFFF + 1 AND wADR <= 16#FFFF THEN
    (* Link Adress *)
    fbJobFc16.bUnitId       := byUnitId;
    fbJobFc16.bFunctionCode := 16;
    fbJobFc16.xIsBoolQuerry := FALSE;
    fbJobFc16.xIsSerialJob  := FALSE;    
    fbJobFc16.metCheckQuerryAdr(wADR,uiQuantity,pWord,wOffset);
END_IF;
END_METHOD

ACTION actFC01:
(* Trig FC1 *)
IF fbJobFc1.xIsLinked AND fbJobFc1.xIsQuerryReady AND NOT fbJobFc1.xIsLocked AND NOT fbJobFc1.xAllJobsDone AND tonDelayRead.Q THEN
    fbJobFc1.metLock();
    xTrigFc1       := TRUE;
    fbTIMEFc1.Start();
ELSIF usiState = 1 AND (NOT fbJobFc1.xIsLinked OR fbJobFc1.xAllJobsDone) THEN
    usiState                := usiState + 1;    
    fbJobFc1.proAllJobsDone := TRUE;
END_IF

(* Send Querry *)
IF usiState = 1 AND xTrigFc1 THEN
	xTrigDelayRead 	:= FALSE;
    ITF_MbPortControllQuerry.metMbTcpClient(    stIp        := scParameter.fbstIp.stValue,
                                                wPort       := scParameter.fbwPort.wValue,
                                                scKeepAlive := scKeepAlive,
                                                tTimeOut    := scParameter.fbtTimeOut.tValue,
                                                utQuery     := fbJobFc1.utQuery,
                                                xTrigger    := xTrigFc1,
                                                utResponse  := fbJobFc1.utResponse,
                                                xError      => xErrorMbClientTcp,
                                                uiID        => uiIdMbClientTcp);       
END_IF;
(* Get Response *) 
IF usiState = 1 AND NOT xTrigFc1 AND fbJobFc1.xIsLocked AND NOT fbJobFc1.xJobDone THEN
    usiState            := usiState + 1;
    ltMessungFc1        := fbTIMEFc1.Stop();
    metCheckOnError(xErrorMbClientTcp);
    fbJobFc1.metCallAfterResponse(xErrorMbClientTcp,uiIdMbClientTcp);
END_IF;
END_ACTION

ACTION actFC03:
(* Trig FC3 *)
IF fbJobFc3.xIsLinked AND fbJobFc3.xIsQuerryReady AND NOT fbJobFc3.xIsLocked AND NOT fbJobFc3.xAllJobsDone AND tonDelayRead.Q THEN
    fbJobFc3.metLock();
    xTrigFc3       := TRUE;
    fbTIMEFc3.Start();
ELSIF usiState = 3 AND (NOT fbJobFc3.xIsLinked OR fbJobFc3.xAllJobsDone) THEN
    usiState                := usiState + 1;    
    fbJobFc3.proAllJobsDone := TRUE;
END_IF

(* Send Querry *)
IF usiState = 3 AND xTrigFc3 THEN
	xTrigDelayRead 	:= FALSE;
    ITF_MbPortControllQuerry.metMbTcpClient(    stIp        := scParameter.fbstIp.stValue,
                                                wPort       := scParameter.fbwPort.wValue,
                                                scKeepAlive := scKeepAlive,
                                                tTimeOut    := scParameter.fbtTimeOut.tValue,
                                                utQuery     := fbJobFc3.utQuery,
                                                xTrigger    := xTrigFc3,
                                                utResponse  := fbJobFc3.utResponse,
                                                xError      => xErrorMbClientTcp,
                                                uiID        => uiIdMbClientTcp);       
END_IF;
(* Get Response *) 
IF usiState = 3 AND NOT xTrigFc3 AND fbJobFc3.xIsLocked AND NOT fbJobFc3.xJobDone THEN
    usiState            := usiState + 1;
    ltMessungFc3        := fbTIMEFc3.Stop();
    metCheckOnError(xErrorMbClientTcp);
    fbJobFc3.metCallAfterResponse(xErrorMbClientTcp,uiIdMbClientTcp);
END_IF;
END_ACTION

ACTION actConfig:
(* Config File *)
fbConfigFile();

scParameter.fbxEnable           (_usiParaNr :=  1, itfConfigFb := fbconfigFile                                           );
scparameter.fbbyUnitId          (_usiParaNr :=  2, itfConfigFb := fbconfigFile , _MinInit := 0      ,_MaxInit := 247     );
scparameter.fbstIp              (_usiParaNr :=  3, itfConfigFb := fbconfigFile );
scparameter.fbwPort             (_usiParaNr :=  4, itfConfigFb := fbconfigFile );
scparameter.fbtTimeOut          (_usiParaNr :=  5, itfConfigFb := fbconfigFile , _MinInit := T#10MS ,_MaxInit := T#10M   );
scparameter.fbtScanRate         (_usiParaNr :=  6, itfConfigFb := fbconfigFile , _MinInit := T#00MS ,_MaxInit := T#10M   );
scparameter.fbxKeepAlive        (_usiParaNr :=  7, itfConfigFb := fbconfigFile );
scparameter.fbtMaxIdleTime      (_usiParaNr :=  8, itfConfigFb := fbconfigFile , _MinInit := T#50MS ,_MaxInit := T#10M   );
scparameter.fbtIntervall        (_usiParaNr :=  9, itfConfigFb := fbconfigFile , _MinInit := T#50MS ,_MaxInit := T#10M   );
scparameter.fbudiProbes         (_usiParaNr := 10, itfConfigFb := fbconfigFile , _MinInit := 0      ,_MaxInit := 50      );
scParameter.fbtDelayRead		(_usiParaNr := 11, itfConfigFb := fbconfigFile , _MinInit := T#1MS  ,_MaxInit := T#10M   );	
scParameter.fbtDelayWrite		(_usiParaNr := 12, itfConfigFb := fbconfigFile , _MinInit := T#1MS  ,_MaxInit := T#10M   );
END_ACTION

ACTION actFC02:
(* Trig FC2 *)
IF fbJobFc2.xIsLinked AND fbJobFc2.xIsQuerryReady AND NOT fbJobFc2.xIsLocked AND NOT fbJobFc2.xAllJobsDone AND tonDelayRead.Q THEN
    fbJobFc2.metLock();
    xTrigFc2       := TRUE;
    fbTIMEFc2.Start();
ELSIF usiState = 2 AND (NOT fbJobFc2.xIsLinked OR fbJobFc2.xAllJobsDone) THEN
    usiState                := usiState + 1;    
    fbJobFc2.proAllJobsDone := TRUE;
END_IF

(* Send Querry *)
IF usiState = 2 AND xTrigFc2 THEN
	xTrigDelayRead 	:= FALSE;
    ITF_MbPortControllQuerry.metMbTcpClient(    stIp        := scParameter.fbstIp.stValue,
                                                wPort       := scParameter.fbwPort.wValue,
                                                scKeepAlive := scKeepAlive,
                                                tTimeOut    := scParameter.fbtTimeOut.tValue,
                                                utQuery     := fbJobFc2.utQuery,
                                                xTrigger    := xTrigFc2,
                                                utResponse  := fbJobFc2.utResponse,
                                                xError      => xErrorMbClientTcp,
                                                uiID        => uiIdMbClientTcp);       
END_IF;
(* Get Response *) 
IF usiState = 2 AND NOT xTrigFc2 AND fbJobFc2.xIsLocked AND NOT fbJobFc2.xJobDone THEN
    usiState            := usiState + 1;
    ltMessungFc2        := fbTIMEFc2.Stop();
    metCheckOnError(xErrorMbClientTcp);
    fbJobFc2.metCallAfterResponse(xErrorMbClientTcp,uiIdMbClientTcp);
END_IF;
END_ACTION

ACTION actFC16:
(* Trig FC16 *)
IF fbJobFc16.xIsLinked AND fbJobFc16.xIsQuerryReady AND NOT fbJobFc16.xIsLocked AND NOT fbJobFc16.xAllJobsDone AND tonDelayWrite.Q  THEN
    fbJobFc16.metLock();
    xTrigFc16       := TRUE;
    fbTIMEFc16.Start();
ELSIF usiState = 8 AND (NOT fbJobFc16.xIsLinked OR fbJobFc16.xAllJobsDone) THEN
    usiState                    := usiState + 1; 
    fbJobFc16.proAllJobsDone    := TRUE;   
END_IF
(* Send Querry *)
IF usiState = 8  AND xTrigFc16 THEN
	xTrigDelayWrite := FALSE;
    ITF_MbPortControllQuerry.metMbTcpClient(    stIp        := scParameter.fbstIp.stValue,
                                                wPort       := scParameter.fbwPort.wValue,
                                                scKeepAlive := scKeepAlive,
                                                tTimeOut    := scParameter.fbtTimeOut.tValue,
                                                utQuery     := fbJobFc16.utQuery,
                                                xTrigger    := xTrigFc16,
                                                utResponse  := fbJobFc16.utResponse,
                                                xError      => xErrorMbClientTcp,
                                                uiID        => uiIdMbClientTcp);       
END_IF;
(* Get Response *) 
IF usiState = 8 AND NOT xTrigFc16 AND fbJobFc16.xIsLocked AND NOT fbJobFc16.xJobDone THEN
    usiState             := usiState + 1;
    ltMessungFc16        := fbTIMEFc16.Stop();
    metCheckOnError(xErrorMbClientTcp);
    fbJobFc16.metCallAfterResponse(xErrorMbClientTcp,uiIdMbClientTcp);
END_IF;
END_ACTION

PROPERTY proNodeReference : REFERENCE TO fbMbTcpClient
GET
proNodeReference REF= THIS^;
END_GET
END_PROPERTY

ACTION actFC43:
(* Trig FC43 *)
IF usiState = 9 AND NOT xDoneFc43 AND NOT xActiveFc43 THEN
	xTrigFc43       	:= TRUE;
	xActiveFc43			:= TRUE;
	tTimeOutFc43		:= T#1S;
	utIdentifyQuerry.bUnitId			:= byUnitId;
	utIdentifyQuerry.bFunctionCode		:= 43;	
	utIdentifyQuerry.IIdentifyObject	:= fbIdentifyObject;	
    fbTIMEFc43.Start();
ELSIF usiState = 9 AND NOT xActiveFc43 THEN
    usiState                := usiState + 1; 
END_IF
(* Send Querry *)
IF usiState = 9 AND xTrigFc43 THEN											
    ITF_MbPortControllQuerry.metMbTcpClient(    stIp        := scParameter.fbstIp.stValue,
                                                wPort       := scParameter.fbwPort.wValue,
                                                scKeepAlive := scKeepAlive,
                                                tTimeOut    := tTimeOutFc43,
                                                utQuery     := utIdentifyQuerry,
                                                xTrigger    := xTrigFc43,
                                                utResponse  := utIdentifyResponse,
                                                xError      => xErrorMbClientTcp,
                                                uiID        => uiIdMbClientTcp);    
END_IF;
(* Get Response *) 
IF usiState = 9 AND NOT xTrigFc43 AND xActiveFc43 AND NOT xDoneFc43 THEN
    usiState            := usiState + 1;
    ltMessungFc43       := fbTIMEFc43.Stop();
	xActiveFc43 		:= FALSE;
	IF uiIdMbClientTcp = 16#99 THEN
		xDoneFc43			:= FALSE;
	ELSE
		xDoneFc43			:= TRUE;
	END_IF;
END_IF;
END_ACTION

{attribute 'monitoring' := 'call'}
PROPERTY sMajorMinorRevision : STRING(WagoAppPlcModbus.Parameter.MAX_IDENTIFICATION_MEMBER_LENGTH)
GET
sMajorMinorRevision := fbIdentifyObject.sMajorMinorRevision;
END_GET
END_PROPERTY

{attribute 'monitoring' := 'call'}
PROPERTY sProductCode : STRING(WagoAppPlcModbus.Parameter.MAX_IDENTIFICATION_MEMBER_LENGTH)
GET
sProductCode := fbIdentifyObject.sProductCode;
END_GET
END_PROPERTY

{attribute 'monitoring' := 'call'}
PROPERTY sVendorName : STRING(WagoAppPlcModbus.Parameter.MAX_IDENTIFICATION_MEMBER_LENGTH)
GET
sVendorName := fbIdentifyObject.sVendorName;
END_GET
END_PROPERTY

PROPERTY proModBusOK : BOOL
GET
proModBusOK := xComAktive AND NOT xError;
END_GET
END_PROPERTY

METHOD FINAL metFc5WriteCoil
VAR_INPUT
    wADR                :   WORD;
    pByte               :   POINTER TO BYTE;
    uiQuantity          :   UINT;               // Anzahl Coils Max 2000   
    wOffset             :   WORD;               // Pointer Offset wenn BOOL Array > 125     
END_VAR
VAR
    diCurrentJop        :   DINT;
    uiFor               :   UINT;
    usiCountWords       :   UINT;
    wTempValue          :   WORD;    
END_VAR
(* Limit Write Multiple Coil *)
uiQuantity := LIMIT(1,uiQuantity,1);
(* Check if valid Pointer and Adress *)
IF pByte <> 0 AND wOffset + uiQuantity <= 16#FFFF + 1 AND wADR <= 16#FFFF THEN
    (* Link Adress *)
    fbJobFc5.bUnitId       := byUnitId;
    fbJobFc5.bFunctionCode := 5;
    fbJobFc5.xIsBoolQuerry := TRUE;
    fbJobFc5.xIsSerialJob  := TRUE;           
    fbJobFc5.metCheckQuerryAdr(wADR,uiQuantity,pByte,wOffset);    
END_IF;
END_METHOD

METHOD FINAL metFc6WriteHoldingRegister
VAR_INPUT
    wADR                :   WORD;
    pWord               :   POINTER TO WORD;
    uiQuantity          :   UINT;               // Anzahl Words Max 125
    wOffset             :   WORD;               // Pointer Offset wenn Array > 125 WORD    
END_VAR
VAR
    diCurrentJop        :   DINT;
    uiFor               :   UINT;
END_VAR
(* Limit Write Holding Registers *)
uiQuantity := LIMIT(1,uiQuantity,1);
(* Check if valid Pointer and Adress *)
IF pWord <> 0 AND wOffset + uiQuantity <= 16#FFFF + 1 AND wADR <= 16#FFFF THEN
    (* Link Adress *)
    fbJobFc6.bUnitId       := byUnitId;
    fbJobFc6.bFunctionCode := 6;
    fbJobFc6.xIsBoolQuerry := FALSE;
    fbJobFc6.xIsSerialJob  := FALSE;        
    fbJobFc6.metCheckQuerryAdr(wADR,uiQuantity,pWord,wOffset);
END_IF;
END_METHOD

ACTION actFC05:
(* Trig FC1 *)
IF fbJobFc5.xIsLinked AND fbJobFc5.xIsQuerryReady AND NOT fbJobFc5.xIsLocked AND NOT fbJobFc5.xAllJobsDone AND tonDelayWrite.Q THEN
    fbJobFc5.metLock();
    xTrigFc5       := TRUE;
    fbTIMEFc5.Start();
ELSIF usiState = 5 AND (NOT fbJobFc5.xIsLinked OR fbJobFc5.xAllJobsDone) THEN
    usiState                    := usiState + 1; 
    fbJobFc5.proAllJobsDone    := TRUE;   
END_IF;

(* Send Querry *)
IF usiState = 5 AND xTrigFc5 THEN
	xTrigDelayWrite := FALSE;
    ITF_MbPortControllQuerry.metMbTcpClient(    stIp        := scParameter.fbstIp.stValue,
                                                wPort       := scParameter.fbwPort.wValue,
                                                scKeepAlive := scKeepAlive,
                                                tTimeOut    := scParameter.fbtTimeOut.tValue,
                                                utQuery     := fbJobFc5.utQuery,
                                                xTrigger    := xTrigFc5,
                                                utResponse  := fbJobFc5.utResponse,
                                                xError      => xErrorMbClientTcp,
                                                uiID        => uiIdMbClientTcp);  
END_IF;
(* Get Response *) 
IF -usiState = 5 AND NOT xTrigFc5 AND fbJobFc5.xIsLocked AND NOT fbJobFc5.xJobDone  THEN 
    usiState            := usiState + 1;
    ltMessungFc5       := fbTIMEFc5.Stop();
    metCheckOnError(xErrorMbClientTcp);
    fbJobFc5.metCallAfterResponse(xErrorMbClientTcp,uiIdMbClientTcp);
END_IF;
END_ACTION

ACTION actFC06:
(* Trig FC6 *)
IF fbJobFc6.xIsLinked AND fbJobFc6.xIsQuerryReady AND NOT fbJobFc6.xIsLocked AND NOT fbJobFc6.xAllJobsDone AND tonDelayWrite.Q  THEN
    fbJobFc6.metLock();
    xTrigFc6       := TRUE;
    fbTIMEFc6.Start();
ELSIF usiState = 6 AND (NOT fbJobFc6.xIsLinked OR fbJobFc6.xAllJobsDone) THEN
    usiState                    := usiState + 1; 
    fbJobFc6.proAllJobsDone    := TRUE;   
END_IF;

(* Send Querry *)
IF usiState = 6 AND xTrigFc6 THEN
	xTrigDelayWrite := FALSE;
    ITF_MbPortControllQuerry.metMbTcpClient(    stIp        := scParameter.fbstIp.stValue,
                                                wPort       := scParameter.fbwPort.wValue,
                                                scKeepAlive := scKeepAlive,
                                                tTimeOut    := scParameter.fbtTimeOut.tValue,
                                                utQuery     := fbJobFc6.utQuery,
                                                xTrigger    := xTrigFc6,
                                                utResponse  := fbJobFc6.utResponse,
                                                xError      => xErrorMbClientTcp,
                                                uiID        => uiIdMbClientTcp);  											
END_IF;
(* Get Response *) 
IF usiState = 6 AND NOT xTrigFc6 AND fbJobFc6.xIsLocked AND NOT fbJobFc6.xJobDone THEN    
    usiState            := usiState + 1;
    ltMessungFc6        := fbTIMEFc6.Stop();
    metCheckOnError(xErrorMbClientTcp);
    fbJobFc6.metCallAfterResponse(xErrorMbClientTcp,uiIdMbClientTcp);
END_IF;
END_ACTION

PROPERTY proModBusErrorText : String(20)
GET
proModBusErrorText := TO_STRING(MAX(fbJobFc1.eError,fbJobFc2.eError,fbJobFc3.eError,fbJobFc4.eError,fbJobFc5.eError,fbJobFc6.eError,fbJobFc15.eError,fbJobFc16.eError));
END_GET
END_PROPERTY

PROPERTY proModBusEnabled : BOOL
GET
proModBusEnabled := scParameter.fbxEnable.xValue;
END_GET
END_PROPERTY

PROPERTY proITF_BMK : CtaAppBmk.ITF_BMK
GET
proITF_BMK := ITF_BMK;
END_GET
END_PROPERTY

METHOD metITF_BMK
VAR_INPUT
	ITF_BMK_IN : CtaAppBmk.ITF_BMK;
END_VAR
ITF_BMK := ITF_BMK_IN;
END_METHOD

ACTION actDelay:
(* Delay Read *)
tonDelayRead(	IN	:= xTrigDelayRead AND xTrigDelayWrite,
			 	PT 	:= scParameter.fbtDelayRead.proValue);
(* Delay Write *)
tonDelayWrite(	IN	:= xTrigDelayRead AND xTrigDelayWrite,
			 	PT 	:= scParameter.fbtDelayWrite.proValue);
				
(* Trig *)
xTrigDelayRead 	:= TRUE;
xTrigDelayWrite := TRUE;
END_ACTION

END_FUNCTION_BLOCK

// 21 Interface/NETWORK/ITF_TCP_NODE
INTERFACE ITF_TCP_NODE EXTENDS __SYSTEM.IQueryInterface

PROPERTY proNodeReference : REFERENCE TO fbMbTcpClient
GET
END_GET
END_PROPERTY

END_INTERFACE

// 21 Interface/NETWORK/ITF_MbPortControllTcp
INTERFACE ITF_MbPortControllTcp EXTENDS __SYSTEM.IQueryInterface

METHOD metMbTcpClient
VAR_INPUT
    stIp        : STRING;
    wPort       : WORD;
END_VAR
VAR_IN_OUT
    scKeepAlive : WagoAppPlcModbus.typKeepAlive;
	tTimeOut	: TIME;
	utQuery	    : WagoAppPlcModbus.typMbQuery;
	xTrigger	: BOOL;
	utResponse	: WagoAppPlcModbus.typMbResponse;
END_VAR
VAR_OUTPUT
	xError	: BOOL;
	uiID	: UINT;
END_VAR
END_METHOD

METHOD metSyncClient : BOOL
VAR_IN_OUT
    xAllJobsDone    : BOOL;
    bIdOfCall       : BYTE;
END_VAR
VAR_INPUT
    ITF_TCP_NODE : ITF_TCP_NODE;
END_VAR
END_METHOD

END_INTERFACE

// 30 Program Organization Units/CONVERTER/fcCheckIp
FUNCTION fcCheckIp : BOOL
VAR_INPUT
    stIp           : STRING[20];
END_VAR
VAR
    iFor           : INT;
    iCountPacket   : INT;
    iCountPoint    : INT;
    iCountZiffer   : INT;
    xFail          : BOOL;
END_VAR

FOR iFor := LEN(stIp) TO 0 BY -1 DO
    // Check Termination
    IF iFor = LEN(stIp) THEN
        IF stIp[iFor] <> 0 THEN 
            xFail := TRUE; // No Termination
            EXIT;       
        END_IF;
	ELSE
        // Check if Ziffer
        IF stIp[iFor] >= 48 AND stIp[iFor] <= 57 THEN    
            IF iCountZiffer < 3 THEN
                IF iCountZiffer = 0 THEN
                    IF iFor >= 2 THEN
                        IF stIp[iFor - 2] >= 50 THEN
                            // Check if Ziffer <= 5
                            IF stIp[iFor] <= 53 THEN     
                                iCountZiffer := iCountZiffer + 1;
                            ELSE
                                xFail := TRUE;  // Max is 255
                                EXIT;
                            END_IF;   
                        ELSE
                            iCountZiffer := iCountZiffer + 1;                   
						END_IF;                        
                    ELSE
                        iCountZiffer := iCountZiffer + 1;
					END_IF
                ELSIF iCountZiffer = 1 THEN
                    IF iFor <> 0 THEN
                        IF stIp[iFor - 1] = 46 THEN
                            iCountZiffer := iCountZiffer + 1;
                        // Check if next Ziffer is 2    
                        ELSIF stIp[iFor - 1] >= 50 THEN  
                            // Check if Ziffer <= 5
                            IF stIp[iFor] <= 53 THEN     
                                iCountZiffer := iCountZiffer + 1;
                            ELSE
                                xFail := TRUE;  // Max is 255
                                EXIT;
                            END_IF;    
                        END_IF;
                    ELSE
                        iCountZiffer := iCountZiffer + 1;        
					END_IF;                       
                ELSIF iCountZiffer = 2 THEN
                    IF stIp[iFor] <= 50 THEN
                        iCountZiffer := iCountZiffer + 1;
                    ELSE
                        xFail := TRUE;
                        EXIT;
					END_IF
                END_IF;    
            ELSIF iCountZiffer = 3 THEN
                xFail := TRUE; // More Then 3 Ziffers not allowed!
                EXIT;
            END_IF;
        // Check if Point
        ELSIF stIp[iFor] = 46 THEN
            IF iCountZiffer > 0 THEN
                iCountPacket := iCountPacket + 1;
                iCountPoint  := iCountPoint + 1;
                iCountZiffer := 0;
            ELSE
                xFail := TRUE; // Empty Packet not allowed!
                EXIT;
            END_IF;   
        END_IF;
    END_IF;
END_FOR;

IF xFail THEN
    fcCheckIp := FALSE;
ELSIF iCountPoint = 3 AND iCountPacket = 3 AND iCountZiffer > 0 THEN    
    fcCheckIp := TRUE;
END_IF;

END_FUNCTION

// 30 Program Organization Units/CONVERTER/fcSetInitialIPString
FUNCTION fcSetInitialIPString : BOOL
VAR_INPUT
    ITF_STRING40In : CtaSysConfig.ITF_STRING40;	
END_VAR
VAR
END_VAR

IF __QUERYINTERFACE(ITF_STRING40In,ITF_STRING40In) THEN
    IF ITF_STRING40In.proValue = '' THEN    
        ITF_STRING40In.proValue := '0.0.0.0';
    END_IF;
    fcSetInitialIPString := TRUE;
ELSE
    fcSetInitialIPString := FALSE;
END_IF;

END_FUNCTION

// 21 Interface/NETWORK/ITF_UDP_NODE
INTERFACE ITF_UDP_NODE EXTENDS __SYSTEM.IQueryInterface

PROPERTY proNodeReference : REFERENCE TO fbMbTcpClient
GET
END_GET
END_PROPERTY

END_INTERFACE

// 30 Program Organization Units/CLIENT/NETWORK Client/TCP/fbMbTcpPortControll
FUNCTION_BLOCK fbMbTcpPortControll IMPLEMENTS ITF_MbPortControllTcp
VAR
    fbMbClientTcp               : WagoAppPLCModbus.FbMbMasterTcp;
    bIdOfCourrentCall           : BYTE  := 1;
    bCountetCalls               : BYTE;
    ayNodes                     : ARRAY[1..32] OF ITF_TCP_NODE;
    ayShowNodes                 : ARRAY[1..32] OF BOOL;
END_VAR

METHOD metMbTcpClient
VAR_INPUT
	stIp	: STRING;
	wPort	: WORD;
END_VAR
VAR_IN_OUT
	scKeepAlive	: WagoAppPlcModbus.typKeepAlive;
	tTimeOut	: TIME;
	utQuery	: WagoAppPlcModbus.typMbQuery;
	xTrigger	: BOOL;
	utResponse	: WagoAppPlcModbus.typMbResponse;
END_VAR
VAR_OUTPUT
	xError	: BOOL;
	uiID	: UINT;
END_VAR
VAR
	xDumyTrig	:	BOOL;
END_VAR
IF fbMbClientTcp.xError THEN
	fbMbClientTcp              (xConnect    := FALSE,
								utQuery     := utQuery,
								xTrigger    := xDumyTrig,
								utResponse  := utResponse); 
END_IF;								
fbMbClientTcp              (xConnect    := xTrigger,
                            sHost       := stIp,
                            wPort       := wPort,
                            utKeepAlive := scKeepAlive,
                            eFrameType  := WagoAppPlcModbus.eMbFrameType.ETHERNET,
                            tTimeOut    := tTimeOut,
                            utQuery     := utQuery,
                            xTrigger    := xTrigger,
                            utResponse  := utResponse,
                            xError      => xError); 
							(* Status *)   
                            uiID        := fbMbClientTcp.oStatus.uiID;
END_METHOD

METHOD FINAL metSyncClient : BOOL
VAR_IN_OUT
    xAllJobsDone    : BOOL;
    bIdOfCall       : BYTE;
END_VAR
VAR_INPUT
    ITF_TCP_NODE : ITF_TCP_NODE;
END_VAR
IF bIdOfCall = 0 THEN
    IF bCountetCalls < 32 THEN
        bCountetCalls           := bCountetCalls + 1;
        bIdOfCall               := bCountetCalls;
        ayNodes[bIdOfCall]      := ITF_TCP_NODE;
        ayShowNodes[bIdOfCall]  := __QUERYINTERFACE(ITF_TCP_NODE,ITF_TCP_NODE);
    END_IF;   
END_IF;
IF bIdOfCourrentCall = 0 THEN
    bIdOfCourrentCall := 1;
END_IF;
IF bIdOfCall = bIdOfCourrentCall THEN
    IF xAllJobsDone THEN
        bIdOfCourrentCall := bIdOfCourrentCall + 1;
        IF bIdOfCourrentCall > bCountetCalls THEN
            bIdOfCourrentCall := 1;    
		END_IF
        metSyncClient := FALSE;
    ELSE
        metSyncClient := TRUE;
    END_IF;
END_IF;
END_METHOD

END_FUNCTION_BLOCK

// 30 Program Organization Units/SERVER/ACCES CONTROLL/fbAccesControll
FUNCTION_BLOCK fbAccesControll IMPLEMENTS WagoAppPlcModbus.I_DataAccessListener
VAR_INPUT
    sClientId	    : STRING(20);
END_VAR
VAR_OUTPUT
END_VAR
VAR
    ayACCESBOOL     :   ARRAY[0..4096] OF WORD;
    ayACCESWORD     :   ARRAY[0..4096] OF WORD;
END_VAR

(*

**Function**
	
	This method is called when a anyone wants access to the data model.
	This method have to return with 0 to allow the wanted access.
	Otherwise the access will be rejected by the data model and an
	exception with the return value as error code is send to the client.

**Graphical Illustration**

	.. wago.autoimage::

*)
METHOD beforeAccess : USINT (* error code*)
VAR_INPUT
	(* who is asking*)
	sClientId	: STRING(20);
	(* unit id of the requested data model*)
	bUnitId	: BYTE;
	bFunctionCode	: BYTE;
	wReadAddress	: WORD;
	wReadQuantity	: WORD;
	wWriteAddress	: WORD;
	wWriteQuantity	: WORD;
END_VAR
END_METHOD

(*

**Function**

	This method is called after an access to the data model.
	This method has no return value.

**Graphical Illustration**

	.. wago.autoimage::
	
*)
METHOD afterAccess
VAR_INPUT
	(* who is asking*)
	sClientId	: STRING(20);
	(* unit id of the requested data model*)
	bUnitId	: BYTE;
	bFunctionCode	: BYTE;
	wReadAddress	: WORD;
	wReadQuantity	: WORD;
	wWriteAddress	: WORD;
	wWriteQuantity	: WORD;
	oStatus	: WagoAppPlcModbus.WagoSysErrorBase.FbResult;
END_VAR
END_METHOD

METHOD ALLOWBOOL
VAR_INPUT
    uiAdr   :   UINT;
    xAllow  :   BOOL;
END_VAR
VAR
    uiMod   : UINT;
    uiDiv   : UINT;
END_VAR
uiMod := uiAdr MOD 15;
uiDiv := uiAdr / 15;
IF uiDiv >= TO_UINT(LOWER_BOUND(ayACCESBOOL,1)) AND uiDiv <= TO_UINT(UPPER_BOUND(ayACCESBOOL,1)) THEN    
    IF uiMod    =  0 THEN
        ayACCESBOOL[uiDiv].00 := xAllow;
    ELSIF uiMod =  1 THEN
        ayACCESBOOL[uiDiv].01 := xAllow;
    ELSIF uiMod =  2 THEN
        ayACCESBOOL[uiDiv].02 := xAllow;
    ELSIF uiMod =  3 THEN
        ayACCESBOOL[uiDiv].03 := xAllow;
    ELSIF uiMod =  4 THEN
        ayACCESBOOL[uiDiv].04 := xAllow;
    ELSIF uiMod =  5 THEN
        ayACCESBOOL[uiDiv].05 := xAllow;
    ELSIF uiMod =  6 THEN
        ayACCESBOOL[uiDiv].06 := xAllow;
    ELSIF uiMod =  7 THEN
        ayACCESBOOL[uiDiv].07 := xAllow;
    ELSIF uiMod =  8 THEN
        ayACCESBOOL[uiDiv].08 := xAllow;
    ELSIF uiMod =  9 THEN
        ayACCESBOOL[uiDiv].09 := xAllow;
    ELSIF uiMod = 10 THEN        
        ayACCESBOOL[uiDiv].10 := xAllow;
    ELSIF uiMod = 11 THEN        
        ayACCESBOOL[uiDiv].11 := xAllow;
    ELSIF uiMod = 12 THEN        
        ayACCESBOOL[uiDiv].12 := xAllow;
    ELSIF uiMod = 13 THEN        
        ayACCESBOOL[uiDiv].13 := xAllow;
    ELSIF uiMod = 14 THEN     
        ayACCESBOOL[uiDiv].14 := xAllow;
    ELSIF uiMod = 15 THEN                   
        ayACCESBOOL[uiDiv].15 := xAllow;
    END_IF;
END_IF;
END_METHOD

END_FUNCTION_BLOCK

// 40 Visualizations/SERVER/PARAMETER/TCP/VIS_ModBusParameter_TCP
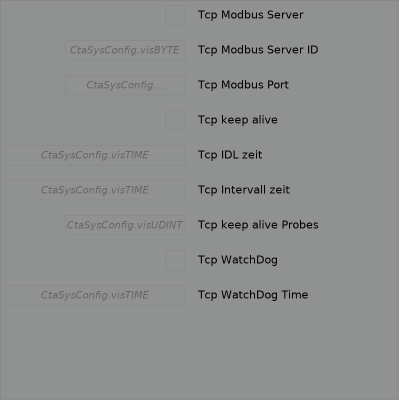
VISUALIZATION VIS_ModBusParameter_TCP  // 399x400
VAR_IN_OUT
    fbModBusServerIn   : fbModBusServer;  
END_VAR
    Label (195,5 195x20), "Tcp Modbus Server"
    Label (195,40 195x20), "Tcp Modbus Server ID"
    Label (195,75 195x20), "Tcp Modbus Port"
    Label (195,110 195x20), "Tcp keep alive"
    Label (195,145 195x20), "Tcp IDL zeit"
    Label (195,180 195x20), "Tcp Intervall zeit"
    Label (195,215 195x20), "Tcp keep alive Probes"
    Label (195,250 195x20), "Tcp WatchDog"
    Label (195,285 195x20), "Tcp WatchDog Time"
    Frame (5,285 180x20)
        shows CtaSysConfig.visTIME(visfbTIMEIn := fbModBusServerIn.scParameter.scTcp.fbtWatchDog)
    Frame (165,250 20x20)
        shows CtaSysConfig.visBOOL(visfbBOOLIn := fbModBusServerIn.scParameter.scTcp.fbxEnableWatchDog)
    Frame (65,215 120x20)
        shows CtaSysConfig.visUDINT(visfbUDINTIn := fbModBusServerIn.scParameter.scTcp.fbudiProbes)
    Frame (5,180 180x20)
        shows CtaSysConfig.visTIME(visfbTIMEIn := fbModBusServerIn.scParameter.scTcp.fbtIntervall)
    Frame (5,145 180x20)
        shows CtaSysConfig.visTIME(visfbTIMEIn := fbModBusServerIn.scParameter.scTcp.fbtMaxIdleTime)
    Frame (165,110 20x20)
        shows CtaSysConfig.visBOOL(visfbBOOLIn := fbModBusServerIn.scParameter.scTcp.fbxKeepAlive)
    Frame (65,75 120x20)
        shows CtaSysConfig.visWORD_DEZ(visfbWORDIn := fbModBusServerIn.scParameter.scTcp.fbwPort)
    Frame (65,40 120x20)
        shows CtaSysConfig.visBYTE(visfbBYTEIn := fbModBusServerIn.scParameter.scTcp.fbbyUnitId)
    Frame (165,5 20x20)
        shows CtaSysConfig.visBOOL(visfbBOOLIn := fbModBusServerIn.scParameter.scTcp.fbxEnable)
END_VISUALIZATION

// 40 Visualizations/SERVER/VIS_ModBusServer
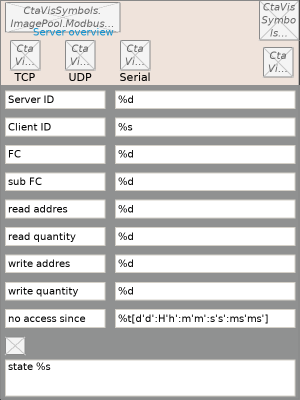
VISUALIZATION VIS_ModBusServer  // 300x400
VAR_IN_OUT
	{attribute 'VAR_IN_OUT_AS_POINTER'}
	fbModBusServerIn   : fbModBusServer;      
END_VAR
VAR
    usiTcpUdpSerial     :   USINT;
END_VAR
    Rectangle (0,0 300x400)
    Rectangle (1,85 299x315)
    Image (5,2 115x30), image: CtaVisSymbols.ImagePool.Modbus_Organization_Logo
    Label (30,27 150x10), "Server overview"
    Image (263,47 30x30), image: CtaVisSymbols.ImagePool.gear
        OnMouseClick:  Dialog=VIS_ModBus_PopUp, Parameters={usiTcpUdpSerial: usiTcpUdpSerial, fbModBusServerIn: fbModBusServerIn}, Selected={0: }, OpenModal=True, OpenCentered=True
    Frame (5,86 290x310), frame switch variable: usiTcpUdpSerial
        shows VIS_ModBusAccesInfo(byServerId := fbModBusServerIn.scParameter.scTcp.fbbyUnitId.byValue, FbMbAccessInfo := fbModBusServerIn.fbMbShowAccesTcp, ltLastAcces := fbModBusServerIn.ltLastAccesTcp, xError := fbModBusServerIn.xErrorTcp, xWatchDogError := fbModBusServerIn.xErrorWatchDogTcp)
        shows VIS_ModBusAccesInfo(byServerId := fbModBusServerIn.scParameter.scUdp.fbbyUnitId.byValue, FbMbAccessInfo := fbModBusServerIn.fbMbShowAccesUdp, ltLastAcces := fbModBusServerIn.ltLastAccesUdp, xError := fbModBusServerIn.xErrorUdp, xWatchDogError := fbModBusServerIn.xErrorWatchDogUdp)
        shows VIS_ModBusAccesInfo(byServerId := fbModBusServerIn.scParameter.scSerial.fbbyUnitId.byValue, FbMbAccessInfo := fbModBusServerIn.fbMbShowAccesSerial, ltLastAcces := fbModBusServerIn.ltLastAccesSerial, xError := fbModBusServerIn.xErrorSerial, xWatchDogError := fbModBusServerIn.xErrorWatchDogSerial)
    Group (115,40 40x45)
        OnMouseClick: execute { usiTcpUdpSerial := 2; }
        Rectangle (0,0 40x44), colour toggle: usiTcpUdpSerial = 2
            OnMouseClick: FrameSelectionChange Selection=SelectedFrame=7903f13b-71ee-407a-abdc-15d9a7e6c2f7, GlobSel=AssignType=Directly, SelType=Locally, SelectionStep=SelectedAction=SwitchNext
        Image (5,0 30x30), image: CtaVisSymbols.ImagePool.lan
            OnMouseClick: FrameSelectionChange Selection=SelectedFrame=7903f13b-71ee-407a-abdc-15d9a7e6c2f7, GlobSel=AssignType=Directly, SelType=Locally, SelectionStep=SelectedAction=SwitchNext
        Label (5,30 30x15), "Serial"
    Group (60,40 40x45)
        OnMouseClick: execute { usiTcpUdpSerial := 1; }
        Rectangle (0,0 40x44), colour toggle: usiTcpUdpSerial = 1
            OnMouseClick: FrameSelectionChange Selection=SelectedFrame=7903f13b-71ee-407a-abdc-15d9a7e6c2f7, Selection=1, GlobSel=AssignType=Directly, SelType=Locally, SelectionStep=SelectedAction=SwitchNext
        Image (5,0 30x30), image: CtaVisSymbols.ImagePool.lan
            OnMouseClick: FrameSelectionChange Selection=SelectedFrame=7903f13b-71ee-407a-abdc-15d9a7e6c2f7, Selection=1, GlobSel=AssignType=Directly, SelType=Locally, SelectionStep=SelectedAction=SwitchNext
        Label (5,30 30x15), "UDP"
    Group (5,40 40x45)
        OnMouseClick: execute { usiTcpUdpSerial := 0; }
        Rectangle (0,0 40x44), colour toggle: usiTcpUdpSerial = 0
            OnMouseClick: FrameSelectionChange Selection=SelectedFrame=7903f13b-71ee-407a-abdc-15d9a7e6c2f7, GlobSel=AssignType=Directly, SelType=Locally, SelectionStep=SelectedAction=SwitchNext
        Image (5,0 30x30), image: CtaVisSymbols.ImagePool.lan
            OnMouseClick: FrameSelectionChange Selection=SelectedFrame=7903f13b-71ee-407a-abdc-15d9a7e6c2f7, GlobSel=AssignType=Directly, SelType=Locally, SelectionStep=SelectedAction=SwitchNext
        Label (5,30 30x15), "TCP"
    Image (259,0 40x40), image: CtaVisSymbols.ImagePool.close_solo_black
        OnMouseClick:  Dialog=Current Dialog, Result=OK, NumpadKeypadSet=True
END_VISUALIZATION

// 40 Visualizations/SERVER/INFO/VIS_ModBusAccesInfo
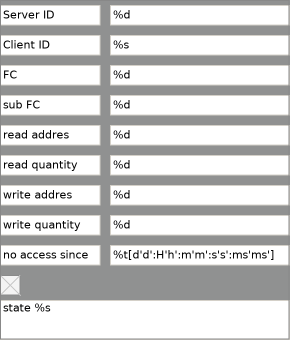
VISUALIZATION VIS_ModBusAccesInfo  // 290x340
VAR_INPUT
    byServerId      :   BYTE;  
	FbMbAccessInfo  :   FbMbAccessInfo;
    ltLastAcces     :   LTIME;
    xError          :   BOOL;
    xWatchDogError  :   BOOL;
END_VAR
    Rectangle (0,0 290x340)
    Textfield (110,35 180x20), "%s", text variable: FbMbAccessInfo.sClientId
    Textfield (110,65 180x20), "%d", text variable: FbMbAccessInfo.bFunctionCode
    Textfield (110,95 180x20), "%d", text variable: FbMbAccessInfo.uiSubFunction
    Textfield (110,125 180x20), "%d", text variable: FbMbAccessInfo.wReadAddress
    Textfield (110,185 180x20), "%d", text variable: FbMbAccessInfo.wWriteAddress
    Textfield (110,215 180x20), "%d", text variable: FbMbAccessInfo.wWriteQuantity
    Textfield (110,155 180x20), "%d", text variable: FbMbAccessInfo.wReadQuantity
    Textfield (0,300 290x40), "state %s", text variable: SEL(xWatchDogError,FbMbAccessInfo.oStatus.GetDescription(),'Error WatchDog')
    Image (0,275 20x20), invisible if: NOT xError, image: CtaVisSymbols.ImagePool.CtaError
    Textfield (0,35 100x20), "Client ID"
    Textfield (0,65 100x20), "FC"
    Textfield (0,95 100x20), "sub FC"
    Textfield (0,125 100x20), "read addres"
    Textfield (0,185 100x20), "write addres"
    Textfield (0,215 100x20), "write quantity"
    Textfield (0,155 100x20), "read quantity"
    Textfield (110,5 180x20), "%d", text variable: byServerId
    Textfield (0,5 100x20), "Server ID"
    Textfield (0,245 100x20), "no access since"
    Textfield (110,245 180x20), "%t[d'd':H'h':m'm':s's':ms'ms']", text variable: ltLastAcces
END_VISUALIZATION

// 40 Visualizations/SERVER/PARAMETER/VIS_ModBus_PopUp
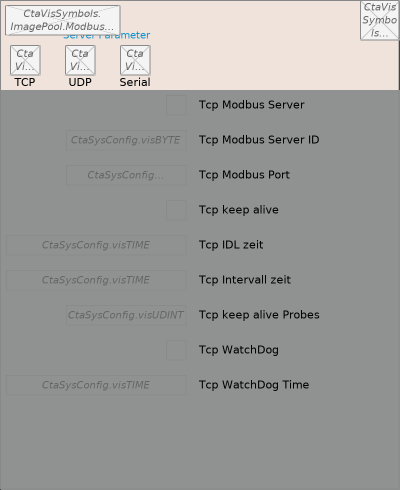
VISUALIZATION VIS_ModBus_PopUp  // 400x490
VAR_IN_OUT
	fbModBusServerIn   : fbModBusServer;  
    {attribute 'VAR_IN_OUT_AS_POINTER'}
    usiTcpUdpSerial    :   USINT;
END_VAR
    Rectangle (0,0 400x490)
    Label (60,30 150x10), "Server Parameter"
    Image (5,5 115x30), image: CtaVisSymbols.ImagePool.Modbus_Organization_Logo
    Group (115,45 40x45)
        OnMouseClick: execute { usiTcpUdpSerial := 2; }
        Rectangle (0,0 40x45), colour toggle: usiTcpUdpSerial = 2
        Image (5,0 30x30), image: CtaVisSymbols.ImagePool.lan
        Label (5,30 30x15), "Serial"
    Group (60,45 40x45)
        OnMouseClick: execute { usiTcpUdpSerial := 1; }
        Rectangle (0,0 40x45), colour toggle: usiTcpUdpSerial = 1
        Image (5,0 30x30), image: CtaVisSymbols.ImagePool.lan
        Label (5,30 30x15), "UDP"
    Group (5,45 40x45)
        OnMouseClick: execute { usiTcpUdpSerial := 0; }
        Rectangle (0,0 40x45), colour toggle: usiTcpUdpSerial = 0
        Image (5,0 30x30), image: CtaVisSymbols.ImagePool.lan
        Label (5,30 30x15), "TCP"
    Frame (1,90 399x400), frame switch variable: usiTcpUdpSerial
        shows VIS_ModBusParameter_TCP(fbModBusServerIn := fbModBusServerIn)
        shows VIS_ModBusParameter_UDP(fbModBusServerIn := fbModBusServerIn)
        shows VIS_ModBusParameter_SERIAL(fbModBusServerIn := fbModBusServerIn)
    Image (360,0 40x40), image: CtaVisSymbols.ImagePool.close_solo_black
        OnMouseClick:  Dialog=VIS_ModBus_PopUp, Result=None, NumpadKeypadSet=True
END_VISUALIZATION

// 40 Visualizations/SERVER/PARAMETER/UDP/VIS_ModBusParameter_UDP
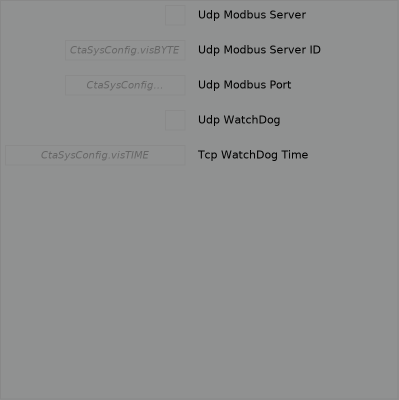
VISUALIZATION VIS_ModBusParameter_UDP  // 399x400
VAR_IN_OUT
    fbModBusServerIn   : fbModBusServer;  
END_VAR
    Label (195,5 195x20), "Udp Modbus Server"
    Label (195,40 195x20), "Udp Modbus Server ID"
    Label (195,75 195x20), "Udp Modbus Port"
    Label (195,110 195x20), "Udp WatchDog"
    Label (195,145 195x20), "Tcp WatchDog Time"
    Frame (5,145 180x20)
        shows CtaSysConfig.visTIME(visfbTIMEIn := fbModBusServerIn.scParameter.scUdp.fbtWatchDog)
    Frame (165,110 20x20)
        shows CtaSysConfig.visBOOL(visfbBOOLIn := fbModBusServerIn.scParameter.scUdp.fbxEnableWatchDog)
    Frame (65,75 120x20)
        shows CtaSysConfig.visWORD_DEZ(visfbWORDIn := fbModBusServerIn.scParameter.scUdp.fbwPort)
    Frame (65,40 120x20)
        shows CtaSysConfig.visBYTE(visfbBYTEIn := fbModBusServerIn.scParameter.scUdp.fbbyUnitId)
    Frame (165,5 20x20)
        shows CtaSysConfig.visBOOL(visfbBOOLIn := fbModBusServerIn.scParameter.scUdp.fbxEnable)
END_VISUALIZATION

// 40 Visualizations/CLIENT/SERIAL Client/SERIAL PORT/VIS_ModBusSerialPort
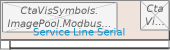
VISUALIZATION VIS_ModBusSerialPort  // 170x50
VAR_IN_OUT
	fbMbSerialPortControllIn   : fbMbSerialPortControll;      
END_VAR
    RoundedRectangle (0,0 170x40)
    Image (1460,183 0x1), image: CtaVisSymbols.ImagePool.ModbusLogo
    Image (2,2 115x30), image: CtaVisSymbols.ImagePool.Modbus_Organization_Logo
    Label (30,27 120x10), "Service Line Serial"
    Image (140,0 30x30), image: CtaVisSymbols.ImagePool.gear
        OnMouseClick:  Dialog=VIS_ModBus_PopUp_Serial_Port_Control, Parameters={fbMbSerialPortControllIn: fbMbSerialPortControllIn}, Selected={0: }, OpenModal=True, OpenCentered=True
    Line (10,50) (10,41), invisible if: fbMbSerialPortControllIn.bCountetCalls < 1
    Line (65,48) (10,48), invisible if: fbMbSerialPortControllIn.bCountetCalls < 1
    Line (170,48) (64,48), invisible if: fbMbSerialPortControllIn.bCountetCalls < 2
END_VISUALIZATION

// 40 Visualizations/CLIENT/NETWORK Client/VIS_ModBusNetworkPortTcp
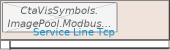
VISUALIZATION VIS_ModBusNetworkPortTcp  // 170x50
VAR_IN_OUT
	fbMbTcpPortControllIn   : fbMbTcpPortControll;      
END_VAR
    RoundedRectangle (0,0 170x40)
    Image (1460,183 0x1), image: CtaVisSymbols.ImagePool.ModbusLogo
    Image (2,2 115x30), image: CtaVisSymbols.ImagePool.Modbus_Organization_Logo
    Label (30,27 120x10), "Service Line Tcp"
    Line (10,50) (10,41), invisible if: fbMbTcpPortControllIn.bCountetCalls < 1
    Line (65,48) (10,48), invisible if: fbMbTcpPortControllIn.bCountetCalls < 1
    Line (170,48) (64,48), invisible if: fbMbTcpPortControllIn.bCountetCalls < 2
END_VISUALIZATION

// 40 Visualizations/HELPER/VIS_IP_INPUT
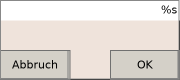
VISUALIZATION VIS_IP_INPUT  // 180x80
VAR_INPUT
    ITF_STRING40In : CtaSysConfig.ITF_STRING40;	
    stIPTemp    :   STRING;
END_VAR
    Rectangle (0,0 180x80)
    Button (110,50 70x30), "OK"
        OnMouseClick: execute {
            IF fcCheckIp(stIPTemp) THEN
                ITF_STRING40In.proValue := stIPTemp;
            ELSE
                ITF_STRING40In.proValue := 'Wrong IP';
            END_IF
        }
        OnMouseClick:  Dialog=VIS_IP_INPUT, Result=OK, NumpadKeypadSet=True
    Button (0,50 70x30), "Abbruch"
        OnMouseClick:  Dialog=VIS_IP_INPUT, Result=Cancel, NumpadKeypadSet=True
    Textfield (0,0 180x20), "%s", text variable: stIPTemp
        OnMouseClick: write the text variable via Default
END_VISUALIZATION

// 40 Visualizations/HELPER/VIS_IP_PARAMETER
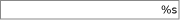
VISUALIZATION VIS_IP_PARAMETER  // 180x20
VAR_INPUT
    ITF_STRING40In : CtaSysConfig.ITF_STRING40;	
END_VAR
    Frame (0,0 180x20), invisible if: NOT __QUERYINTERFACE(ITF_STRING40In,ITF_STRING40In), input disabled if: NOT __QUERYINTERFACE(ITF_STRING40In,ITF_STRING40In)
        shows VIS_IP_PARAMETER_QUERRY(ITF_STRING40In := ITF_STRING40In)
END_VISUALIZATION

// 40 Visualizations/HELPER/VIS_IP_PARAMETER_QUERRY
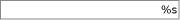
VISUALIZATION VIS_IP_PARAMETER_QUERRY  // 180x20
VAR_INPUT
    ITF_STRING40In : CtaSysConfig.ITF_STRING40;	
END_VAR
    Frame (0,0 180x20), invisible if: NOT __QUERYINTERFACE(ITF_STRING40In,ITF_STRING40In), input disabled if: NOT __QUERYINTERFACE(ITF_STRING40In,ITF_STRING40In)
        shows VIS_IP_PARAMETER_BASE(ITF_STRING40In := ITF_STRING40In)
END_VISUALIZATION

// 40 Visualizations/HELPER/VIS_IP_PARAMETER_BASE
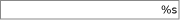
VISUALIZATION VIS_IP_PARAMETER_BASE  // 180x20
VAR_INPUT
    ITF_STRING40In : CtaSysConfig.ITF_STRING40;	
END_VAR
    Textfield (0,0 180x20), "%s", text variable: ITF_STRING40In.proValue, invisible if: NOT fcSetInitialIPString(ITF_STRING40In)
        OnMouseClick:  Dialog=VIS_IP_INPUT, Parameters={stIPTemp: ITF_STRING40In.proValue, ITF_STRING40In: ITF_STRING40In}, OpenModal=True, OpenCentered=True
END_VISUALIZATION

// 40 Visualizations/CLIENT/SERIAL Client/SERIAL Client/VIS_ModBusSerialNode
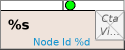
VISUALIZATION VIS_ModBusSerialNode  // 125x50
VAR_INPUT   
	ITF_SERIAL_NODEIN :   ITF_SERIAL_NODE;   
    xCourrentNode     :   BOOL;
END_VAR
    Frame (0,0 125x50), invisible if: NOT __QUERYINTERFACE(ITF_SERIAL_NODEIN,ITF_SERIAL_NODEIN)
        shows VIS_ModBusSerialNode_QUERRY(fbMbSerialClientIn := ITF_SERIAL_NODEIN.proNodeReference)
    Ellipse (65,0 10x10), invisible if: NOT xCourrentNode
END_VISUALIZATION

// 40 Visualizations/CLIENT/SERIAL Client/SERIAL PORT/PARAMETER/VIS_ModBus_PopUp_Serial_Port_Control
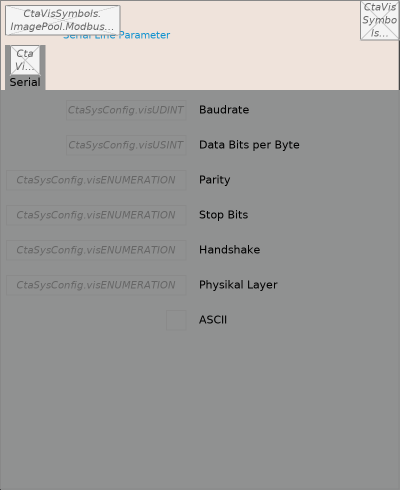
VISUALIZATION VIS_ModBus_PopUp_Serial_Port_Control  // 400x490
VAR_IN_OUT
    {attribute 'VAR_IN_OUT_AS_POINTER'}
	fbMbSerialPortControllIn   : fbMbSerialPortControll;   
END_VAR
    Rectangle (0,0 400x490)
    Label (60,30 150x10), "Serial Line Parameter"
    Image (5,5 115x30), image: CtaVisSymbols.ImagePool.Modbus_Organization_Logo
    Group (5,45 40x45)
        Rectangle (0,0 40x45)
        Image (5,0 30x30), image: CtaVisSymbols.ImagePool.lan
        Label (5,30 30x15), "Serial"
    Frame (1,90 399x400)
        shows VIS_ModBusParameter_Serial_Port_Control(fbMbSerialPortControllIn := fbMbSerialPortControllIn)
        shows VIS_ModBusParameter_UDP(fbModBusServerIn := fbModBusServerIn)
        shows VIS_ModBusParameter_SERIAL(fbModBusServerIn := fbModBusServerIn)
    Image (360,0 40x40), image: CtaVisSymbols.ImagePool.close_solo_black
        OnMouseClick:  Dialog=VIS_ModBus_PopUp_Serial_Port_Control, Result=OK, NumpadKeypadSet=True
END_VISUALIZATION

// 40 Visualizations/CLIENT/SERIAL Client/VIS_SERIAL_LINE_HORIZONTAL
VISUALIZATION VIS_SERIAL_LINE_HORIZONTAL  // 100x4
    Line (100,2) (0,2)
END_VISUALIZATION

// 40 Visualizations/CLIENT/SERIAL Client/SERIAL PORT/PARAMETER/SERIAL/VIS_ModBusParameter_Serial_Port_Control
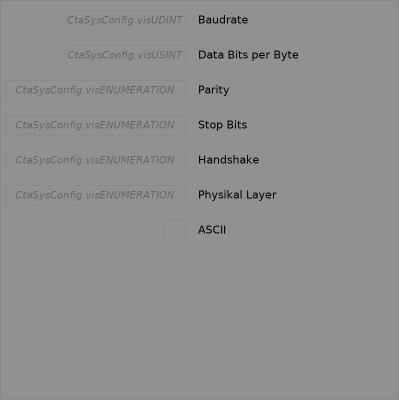
VISUALIZATION VIS_ModBusParameter_Serial_Port_Control  // 399x400
VAR_IN_OUT
    fbMbSerialPortControllIn   : fbMbSerialPortControll;  
END_VAR
    Label (195,10 195x20), "Baudrate"
    Label (195,45 195x20), "Data Bits per Byte"
    Label (195,80 195x20), "Parity"
    Label (195,115 195x20), "Stop Bits"
    Label (195,150 195x20), "Handshake"
    Label (195,185 195x20), "Physikal Layer"
    Label (195,220 195x20), "ASCII"
    Frame (65,10 120x20)
        shows CtaSysConfig.visUDINT(visfbUDINTIn := fbMbSerialPortControllIn.scParameter.fbudiBaudrate)
    Frame (165,220 20x20)
        shows CtaSysConfig.visBOOL(visfbBOOLIn := fbMbSerialPortControllIn.scParameter.fbxRtuOrAscii)
    Frame (5,185 180x20), text list: 'txtPhysikalLayer', text index: CtaSysConfig.fcGetEnumerationId(fbMbSerialPortControllIn.scParameter.fbiPhysikal)
        shows CtaSysConfig.visENUMERATION(visfbENUIn := fbMbSerialPortControllIn.scParameter.fbiPhysikal)
    Frame (5,150 180x20), text list: 'txtHandshake', text index: CtaSysConfig.fcGetEnumerationId(fbMbSerialPortControllIn.scParameter.fbiHandshake)
        shows CtaSysConfig.visENUMERATION(visfbENUIn := fbMbSerialPortControllIn.scParameter.fbiHandshake)
    Frame (5,115 180x20), text list: 'txtStopBits', text index: CtaSysConfig.fcGetEnumerationId(fbMbSerialPortControllIn.scParameter.fbiStopBits)
        shows CtaSysConfig.visENUMERATION(visfbENUIn := fbMbSerialPortControllIn.scParameter.fbiStopBits)
    Frame (5,80 180x20), text list: 'txtParity', text index: CtaSysConfig.fcGetEnumerationId(fbMbSerialPortControllIn.scParameter.fbiParity)
        shows CtaSysConfig.visENUMERATION(visfbENUIn := fbMbSerialPortControllIn.scParameter.fbiParity)
    Frame (65,45 120x20)
        shows CtaSysConfig.visUSINT(visfbUSINTIn := fbMbSerialPortControllIn.scParameter.fbusiDataBits)
END_VISUALIZATION

// 40 Visualizations/CLIENT/SERIAL Client/SERIAL Client/POPUP/VIS_ModBus_Serial_NodePopUp
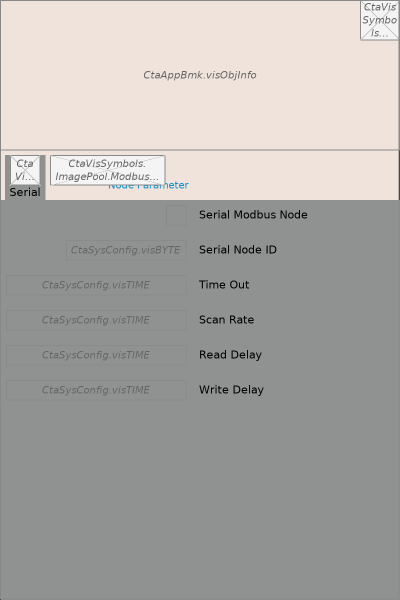
VISUALIZATION VIS_ModBus_Serial_NodePopUp  // 400x600
VAR_IN_OUT
    {attribute 'VAR_IN_OUT_AS_POINTER'}
	fbMbSerialClientIn   : fbMbSerialClient; 
END_VAR
    Rectangle (0,0 400x600)
    Label (105,180 150x10), "Node Parameter"
    Image (50,155 115x30), image: CtaVisSymbols.ImagePool.Modbus_Organization_Logo
    Group (5,155 40x45)
        Rectangle (0,0 40x45)
        Label (5,30 30x15), "Serial"
        Image (5,0 30x30), image: CtaVisSymbols.ImagePool.lan
    Frame (1,200 399x400)
        shows VIS_ModBusParameter_SERIAL_Client(fbMbSerialClientIn := fbMbSerialClientIn)
        shows VIS_ModBusParameter_UDP(fbModBusServerIn := fbModBusServerIn)
        shows VIS_ModBusParameter_SERIAL(fbModBusServerIn := fbModBusServerIn)
    Image (360,0 40x40), image: CtaVisSymbols.ImagePool.close_solo_black
        OnMouseClick:  Dialog=VIS_ModBus_Serial_NodePopUp, Result=OK, NumpadKeypadSet=True
    Frame (0,0 400x150)
        shows CtaAppBmk.visObjInfo(ITF_BMK_IN := fbMbSerialClientIn.proITF_BMK)
END_VISUALIZATION

// 40 Visualizations/CLIENT/SERIAL Client/VIS_SERIAL_LINE_VERTIKAL
VISUALIZATION VIS_SERIAL_LINE_VERTIKAL  // 4x100
    Line (2,0) (2,100)
END_VISUALIZATION

// 40 Visualizations/CLIENT/SERIAL Client/VIS_MODBUS_SERIAL_LINE
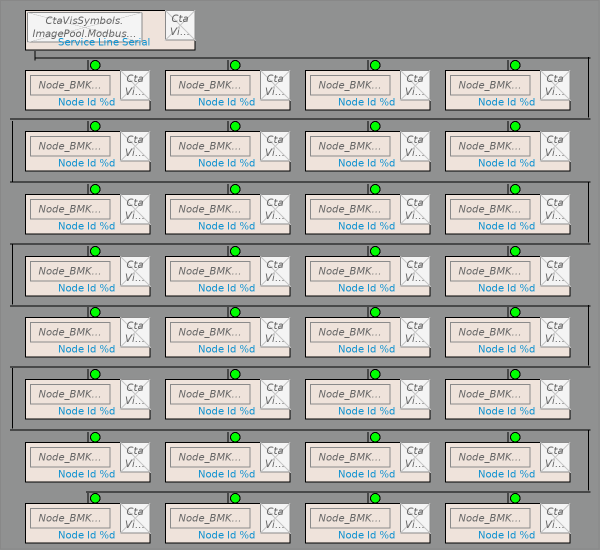
VISUALIZATION VIS_MODBUS_SERIAL_LINE  // 600x550
VAR_IN_OUT
	fbMbSerialPortControllIn   : fbMbSerialPortControll;      
END_VAR
    Frame (509,56 81x4), invisible if: fbMbSerialPortControllIn.bCountetCalls < 5
        shows VIS_SERIAL_LINE_HORIZONTAL()
    Frame (369,56 141x4), invisible if: fbMbSerialPortControllIn.bCountetCalls < 4
        shows VIS_SERIAL_LINE_HORIZONTAL()
    Frame (25,10 170x50)
        shows VIS_ModBusSerialPort(fbMbSerialPortControllIn := fbMbSerialPortControllIn)
    Frame (194,56 36x4), invisible if: fbMbSerialPortControllIn.bCountetCalls < 2
        shows VIS_SERIAL_LINE_HORIZONTAL()
    Frame (586,57 4x60), invisible if: fbMbSerialPortControllIn.bCountetCalls < 5
        shows VIS_SERIAL_LINE_VERTIKAL()
    Frame (10,121 4x60), invisible if: fbMbSerialPortControllIn.bCountetCalls < 9
        shows VIS_SERIAL_LINE_VERTIKAL()
    Frame (10,180 80x4), invisible if: fbMbSerialPortControllIn.bCountetCalls < 9
        shows VIS_SERIAL_LINE_HORIZONTAL()
    Frame (586,182 4x60), invisible if: fbMbSerialPortControllIn.bCountetCalls < 13
        shows VIS_SERIAL_LINE_VERTIKAL()
    Frame (10,244 4x60), invisible if: fbMbSerialPortControllIn.bCountetCalls < 17
        shows VIS_SERIAL_LINE_VERTIKAL()
    Frame (586,305 4x60), invisible if: fbMbSerialPortControllIn.bCountetCalls < 21
        shows VIS_SERIAL_LINE_VERTIKAL()
    Frame (10,368 4x60), invisible if: fbMbSerialPortControllIn.bCountetCalls < 25
        shows VIS_SERIAL_LINE_VERTIKAL()
    Frame (586,430 4x60), invisible if: fbMbSerialPortControllIn.bCountetCalls < 29
        shows VIS_SERIAL_LINE_VERTIKAL()
    Frame (229,56 141x4), invisible if: fbMbSerialPortControllIn.bCountetCalls < 3
        shows VIS_SERIAL_LINE_HORIZONTAL()
    Frame (506,117 84x4), invisible if: fbMbSerialPortControllIn.bCountetCalls < 5
        shows VIS_SERIAL_LINE_HORIZONTAL()
    Frame (366,117 141x4), invisible if: fbMbSerialPortControllIn.bCountetCalls < 6
        shows VIS_SERIAL_LINE_HORIZONTAL()
    Frame (86,117 141x4), invisible if: fbMbSerialPortControllIn.bCountetCalls < 8
        shows VIS_SERIAL_LINE_HORIZONTAL()
    Frame (226,117 141x4), invisible if: fbMbSerialPortControllIn.bCountetCalls < 7
        shows VIS_SERIAL_LINE_HORIZONTAL()
    Frame (10,117 77x4), invisible if: fbMbSerialPortControllIn.bCountetCalls < 9
        shows VIS_SERIAL_LINE_HORIZONTAL()
    Frame (89,180 141x4), invisible if: fbMbSerialPortControllIn.bCountetCalls < 10
        shows VIS_SERIAL_LINE_HORIZONTAL()
    Frame (229,180 141x4), invisible if: fbMbSerialPortControllIn.bCountetCalls < 11
        shows VIS_SERIAL_LINE_HORIZONTAL()
    Frame (509,180 81x4), invisible if: fbMbSerialPortControllIn.bCountetCalls < 13
        shows VIS_SERIAL_LINE_HORIZONTAL()
    Frame (369,180 141x4), invisible if: fbMbSerialPortControllIn.bCountetCalls < 12
        shows VIS_SERIAL_LINE_HORIZONTAL()
    Frame (506,242 84x4), invisible if: fbMbSerialPortControllIn.bCountetCalls < 13
        shows VIS_SERIAL_LINE_HORIZONTAL()
    Frame (366,242 141x4), invisible if: fbMbSerialPortControllIn.bCountetCalls < 14
        shows VIS_SERIAL_LINE_HORIZONTAL()
    Frame (86,242 141x4), invisible if: fbMbSerialPortControllIn.bCountetCalls < 16
        shows VIS_SERIAL_LINE_HORIZONTAL()
    Frame (226,242 141x4), invisible if: fbMbSerialPortControllIn.bCountetCalls < 15
        shows VIS_SERIAL_LINE_HORIZONTAL()
    Frame (10,242 77x4), invisible if: fbMbSerialPortControllIn.bCountetCalls < 17
        shows VIS_SERIAL_LINE_HORIZONTAL()
    Frame (10,304 80x4), invisible if: fbMbSerialPortControllIn.bCountetCalls < 17
        shows VIS_SERIAL_LINE_HORIZONTAL()
    Frame (89,304 141x4), invisible if: fbMbSerialPortControllIn.bCountetCalls < 18
        shows VIS_SERIAL_LINE_HORIZONTAL()
    Frame (229,304 141x4), invisible if: fbMbSerialPortControllIn.bCountetCalls < 19
        shows VIS_SERIAL_LINE_HORIZONTAL()
    Frame (509,304 81x4), invisible if: fbMbSerialPortControllIn.bCountetCalls < 21
        shows VIS_SERIAL_LINE_HORIZONTAL()
    Frame (369,304 141x4), invisible if: fbMbSerialPortControllIn.bCountetCalls < 20
        shows VIS_SERIAL_LINE_HORIZONTAL()
    Frame (506,365 84x4), invisible if: fbMbSerialPortControllIn.bCountetCalls < 21
        shows VIS_SERIAL_LINE_HORIZONTAL()
    Frame (366,365 141x4), invisible if: fbMbSerialPortControllIn.bCountetCalls < 22
        shows VIS_SERIAL_LINE_HORIZONTAL()
    Frame (86,365 141x4), invisible if: fbMbSerialPortControllIn.bCountetCalls < 24
        shows VIS_SERIAL_LINE_HORIZONTAL()
    Frame (226,365 141x4), invisible if: fbMbSerialPortControllIn.bCountetCalls < 23
        shows VIS_SERIAL_LINE_HORIZONTAL()
    Frame (10,365 77x4), invisible if: fbMbSerialPortControllIn.bCountetCalls < 25
        shows VIS_SERIAL_LINE_HORIZONTAL()
    Frame (10,428 80x4), invisible if: fbMbSerialPortControllIn.bCountetCalls < 25
        shows VIS_SERIAL_LINE_HORIZONTAL()
    Frame (89,428 141x4), invisible if: fbMbSerialPortControllIn.bCountetCalls < 26
        shows VIS_SERIAL_LINE_HORIZONTAL()
    Frame (229,428 141x4), invisible if: fbMbSerialPortControllIn.bCountetCalls < 27
        shows VIS_SERIAL_LINE_HORIZONTAL()
    Frame (509,428 81x4), invisible if: fbMbSerialPortControllIn.bCountetCalls < 29
        shows VIS_SERIAL_LINE_HORIZONTAL()
    Frame (369,428 141x4), invisible if: fbMbSerialPortControllIn.bCountetCalls < 28
        shows VIS_SERIAL_LINE_HORIZONTAL()
    Frame (506,490 84x4), invisible if: fbMbSerialPortControllIn.bCountetCalls < 29
        shows VIS_SERIAL_LINE_HORIZONTAL()
    Frame (366,490 141x4), invisible if: fbMbSerialPortControllIn.bCountetCalls < 30
        shows VIS_SERIAL_LINE_HORIZONTAL()
    Frame (86,490 141x4), invisible if: fbMbSerialPortControllIn.bCountetCalls < 32
        shows VIS_SERIAL_LINE_HORIZONTAL()
    Frame (226,490 141x4), invisible if: fbMbSerialPortControllIn.bCountetCalls < 31
        shows VIS_SERIAL_LINE_HORIZONTAL()
    Frame (25,60 125x50), invisible if: NOT fbMbSerialPortControllIn.ayShowNodes[1]
        shows VIS_ModBusSerialNode(ITF_SERIAL_NODEIN := fbMbSerialPortControllIn.ayNodes[1], xCourrentNode := fbMbSerialPortControllIn.bIdOfCourrentCall = 1)
    Frame (305,60 125x50), invisible if: NOT fbMbSerialPortControllIn.ayShowNodes[3]
        shows VIS_ModBusSerialNode(ITF_SERIAL_NODEIN := fbMbSerialPortControllIn.ayNodes[3], xCourrentNode := fbMbSerialPortControllIn.bIdOfCourrentCall = 3)
    Frame (445,60 125x50), invisible if: NOT fbMbSerialPortControllIn.ayShowNodes[4]
        shows VIS_ModBusSerialNode(ITF_SERIAL_NODEIN := fbMbSerialPortControllIn.ayNodes[4], xCourrentNode := fbMbSerialPortControllIn.bIdOfCourrentCall = 4)
    Frame (445,184 125x50), invisible if: NOT fbMbSerialPortControllIn.ayShowNodes[12]
        shows VIS_ModBusSerialNode(ITF_SERIAL_NODEIN := fbMbSerialPortControllIn.ayNodes[12], xCourrentNode := fbMbSerialPortControllIn.bIdOfCourrentCall = 12)
    Frame (25,184 125x50), invisible if: NOT fbMbSerialPortControllIn.ayShowNodes[9]
        shows VIS_ModBusSerialNode(ITF_SERIAL_NODEIN := fbMbSerialPortControllIn.ayNodes[9], xCourrentNode := fbMbSerialPortControllIn.bIdOfCourrentCall = 9)
    Frame (165,184 125x50), invisible if: NOT fbMbSerialPortControllIn.ayShowNodes[10]
        shows VIS_ModBusSerialNode(ITF_SERIAL_NODEIN := fbMbSerialPortControllIn.ayNodes[10], xCourrentNode := fbMbSerialPortControllIn.bIdOfCourrentCall = 10)
    Frame (305,184 125x50), invisible if: NOT fbMbSerialPortControllIn.ayShowNodes[11]
        shows VIS_ModBusSerialNode(ITF_SERIAL_NODEIN := fbMbSerialPortControllIn.ayNodes[11], xCourrentNode := fbMbSerialPortControllIn.bIdOfCourrentCall = 11)
    Frame (25,369 125x50), invisible if: NOT fbMbSerialPortControllIn.ayShowNodes[24]
        shows VIS_ModBusSerialNode(ITF_SERIAL_NODEIN := fbMbSerialPortControllIn.ayNodes[24], xCourrentNode := fbMbSerialPortControllIn.bIdOfCourrentCall = 24)
    Frame (165,369 125x50), invisible if: NOT fbMbSerialPortControllIn.ayShowNodes[23]
        shows VIS_ModBusSerialNode(ITF_SERIAL_NODEIN := fbMbSerialPortControllIn.ayNodes[23], xCourrentNode := fbMbSerialPortControllIn.bIdOfCourrentCall = 23)
    Frame (305,369 125x50), invisible if: NOT fbMbSerialPortControllIn.ayShowNodes[22]
        shows VIS_ModBusSerialNode(ITF_SERIAL_NODEIN := fbMbSerialPortControllIn.ayNodes[22], xCourrentNode := fbMbSerialPortControllIn.bIdOfCourrentCall = 22)
    Frame (445,369 125x50), invisible if: NOT fbMbSerialPortControllIn.ayShowNodes[21]
        shows VIS_ModBusSerialNode(ITF_SERIAL_NODEIN := fbMbSerialPortControllIn.ayNodes[21], xCourrentNode := fbMbSerialPortControllIn.bIdOfCourrentCall = 21)
    Frame (445,432 125x50), invisible if: NOT fbMbSerialPortControllIn.ayShowNodes[28]
        shows VIS_ModBusSerialNode(ITF_SERIAL_NODEIN := fbMbSerialPortControllIn.ayNodes[28], xCourrentNode := fbMbSerialPortControllIn.bIdOfCourrentCall = 28)
    Frame (25,432 125x50), invisible if: NOT fbMbSerialPortControllIn.ayShowNodes[25]
        shows VIS_ModBusSerialNode(ITF_SERIAL_NODEIN := fbMbSerialPortControllIn.ayNodes[25], xCourrentNode := fbMbSerialPortControllIn.bIdOfCourrentCall = 25)
    Frame (165,432 125x50), invisible if: NOT fbMbSerialPortControllIn.ayShowNodes[26]
        shows VIS_ModBusSerialNode(ITF_SERIAL_NODEIN := fbMbSerialPortControllIn.ayNodes[26], xCourrentNode := fbMbSerialPortControllIn.bIdOfCourrentCall = 26)
    Frame (305,432 125x50), invisible if: NOT fbMbSerialPortControllIn.ayShowNodes[27]
        shows VIS_ModBusSerialNode(ITF_SERIAL_NODEIN := fbMbSerialPortControllIn.ayNodes[27], xCourrentNode := fbMbSerialPortControllIn.bIdOfCourrentCall = 27)
    Frame (25,493 125x50), invisible if: NOT fbMbSerialPortControllIn.ayShowNodes[32]
        shows VIS_ModBusSerialNode(ITF_SERIAL_NODEIN := fbMbSerialPortControllIn.ayNodes[32], xCourrentNode := fbMbSerialPortControllIn.bIdOfCourrentCall = 32)
    Frame (165,493 125x50), invisible if: NOT fbMbSerialPortControllIn.ayShowNodes[31]
        shows VIS_ModBusSerialNode(ITF_SERIAL_NODEIN := fbMbSerialPortControllIn.ayNodes[31], xCourrentNode := fbMbSerialPortControllIn.bIdOfCourrentCall = 31)
    Frame (305,493 125x50), invisible if: NOT fbMbSerialPortControllIn.ayShowNodes[30]
        shows VIS_ModBusSerialNode(ITF_SERIAL_NODEIN := fbMbSerialPortControllIn.ayNodes[30], xCourrentNode := fbMbSerialPortControllIn.bIdOfCourrentCall = 30)
    Frame (445,493 125x50), invisible if: NOT fbMbSerialPortControllIn.ayShowNodes[29]
        shows VIS_ModBusSerialNode(ITF_SERIAL_NODEIN := fbMbSerialPortControllIn.ayNodes[29], xCourrentNode := fbMbSerialPortControllIn.bIdOfCourrentCall = 29)
    Frame (165,60 125x50), invisible if: NOT fbMbSerialPortControllIn.ayShowNodes[2]
        shows VIS_ModBusSerialNode(ITF_SERIAL_NODEIN := fbMbSerialPortControllIn.ayNodes[2], xCourrentNode := fbMbSerialPortControllIn.bIdOfCourrentCall = 2)
    Frame (445,121 125x50), invisible if: NOT fbMbSerialPortControllIn.ayShowNodes[5]
        shows VIS_ModBusSerialNode(ITF_SERIAL_NODEIN := fbMbSerialPortControllIn.ayNodes[5], xCourrentNode := fbMbSerialPortControllIn.bIdOfCourrentCall = 5)
    Frame (165,121 125x50), invisible if: NOT fbMbSerialPortControllIn.ayShowNodes[7]
        shows VIS_ModBusSerialNode(ITF_SERIAL_NODEIN := fbMbSerialPortControllIn.ayNodes[7], xCourrentNode := fbMbSerialPortControllIn.bIdOfCourrentCall = 7)
    Frame (25,121 125x50), invisible if: NOT fbMbSerialPortControllIn.ayShowNodes[8]
        shows VIS_ModBusSerialNode(ITF_SERIAL_NODEIN := fbMbSerialPortControllIn.ayNodes[8], xCourrentNode := fbMbSerialPortControllIn.bIdOfCourrentCall = 8)
    Frame (305,121 125x50), invisible if: NOT fbMbSerialPortControllIn.ayShowNodes[6]
        shows VIS_ModBusSerialNode(ITF_SERIAL_NODEIN := fbMbSerialPortControllIn.ayNodes[6], xCourrentNode := fbMbSerialPortControllIn.bIdOfCourrentCall = 6)
    Frame (445,246 125x50), invisible if: NOT fbMbSerialPortControllIn.ayShowNodes[13]
        shows VIS_ModBusSerialNode(ITF_SERIAL_NODEIN := fbMbSerialPortControllIn.ayNodes[13], xCourrentNode := fbMbSerialPortControllIn.bIdOfCourrentCall = 13)
    Frame (305,246 125x50), invisible if: NOT fbMbSerialPortControllIn.ayShowNodes[14]
        shows VIS_ModBusSerialNode(ITF_SERIAL_NODEIN := fbMbSerialPortControllIn.ayNodes[14], xCourrentNode := fbMbSerialPortControllIn.bIdOfCourrentCall = 14)
    Frame (165,246 125x50), invisible if: NOT fbMbSerialPortControllIn.ayShowNodes[15]
        shows VIS_ModBusSerialNode(ITF_SERIAL_NODEIN := fbMbSerialPortControllIn.ayNodes[15], xCourrentNode := fbMbSerialPortControllIn.bIdOfCourrentCall = 15)
    Frame (25,246 125x50), invisible if: NOT fbMbSerialPortControllIn.ayShowNodes[16]
        shows VIS_ModBusSerialNode(ITF_SERIAL_NODEIN := fbMbSerialPortControllIn.ayNodes[16], xCourrentNode := fbMbSerialPortControllIn.bIdOfCourrentCall = 16)
    Frame (25,307 125x50), invisible if: NOT fbMbSerialPortControllIn.ayShowNodes[17]
        shows VIS_ModBusSerialNode(ITF_SERIAL_NODEIN := fbMbSerialPortControllIn.ayNodes[17], xCourrentNode := fbMbSerialPortControllIn.bIdOfCourrentCall = 17)
    Frame (445,307 125x50), invisible if: NOT fbMbSerialPortControllIn.ayShowNodes[20]
        shows VIS_ModBusSerialNode(ITF_SERIAL_NODEIN := fbMbSerialPortControllIn.ayNodes[20], xCourrentNode := fbMbSerialPortControllIn.bIdOfCourrentCall = 20)
    Frame (165,307 125x50), invisible if: NOT fbMbSerialPortControllIn.ayShowNodes[18]
        shows VIS_ModBusSerialNode(ITF_SERIAL_NODEIN := fbMbSerialPortControllIn.ayNodes[18], xCourrentNode := fbMbSerialPortControllIn.bIdOfCourrentCall = 18)
    Frame (305,307 125x50), invisible if: NOT fbMbSerialPortControllIn.ayShowNodes[19]
        shows VIS_ModBusSerialNode(ITF_SERIAL_NODEIN := fbMbSerialPortControllIn.ayNodes[19], xCourrentNode := fbMbSerialPortControllIn.bIdOfCourrentCall = 19)
END_VISUALIZATION

// 40 Visualizations/CLIENT/SERIAL Client/SERIAL Client/VIS_ModBusSerialNode_QUERRY
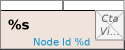
VISUALIZATION VIS_ModBusSerialNode_QUERRY  // 125x50
VAR_IN_OUT
	fbMbSerialClientIn   : REFERENCE TO fbMbSerialClient;      
END_VAR
    RoundedRectangle (0,10 125x40), colour toggle: fbMbSerialClientIn.xError
    RoundedRectangle (0,10 125x40), colour toggle: fbMbSerialClientIn.xError, invisible if: fbMbSerialClientIn.xComAktive
    Image (95,10 30x30), image: CtaVisSymbols.ImagePool.gear
        OnMouseClick:  Dialog=VIS_ModBus_Serial_NodePopUp, Parameters={fbMbSerialClientIn: fbMbSerialClientIn}, Selected={0: }, OpenModal=True, OpenCentered=True
    Textfield (30,37 90x10), "Node Id %d", text variable: fbMbSerialClientIn.byUnitId, invisible if: NOT __ISVALIDREF(fbMbSerialClientIn)
    Line (63,10) (63,0)
    Frame (5,15 80x20)
        shows Node_BMK(ITF_BMK := fbMbSerialClientIn.proITF_BMK)
END_VISUALIZATION

// 40 Visualizations/SERVER/PARAMETER/SERIAL/VIS_ModBusParameter_SERIAL
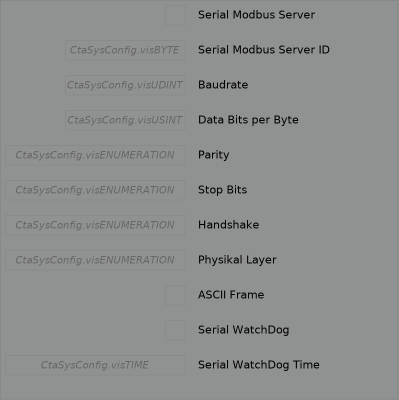
VISUALIZATION VIS_ModBusParameter_SERIAL  // 399x400
VAR_IN_OUT
    fbModBusServerIn   : fbModBusServer;  
END_VAR
    Label (195,5 195x20), "Serial Modbus Server"
    Label (195,40 195x20), "Serial Modbus Server ID"
    Label (195,75 195x20), "Baudrate"
    Label (195,110 195x20), "Data Bits per Byte"
    Label (195,145 195x20), "Parity"
    Label (195,180 195x20), "Stop Bits"
    Label (195,215 195x20), "Handshake"
    Label (195,250 195x20), "Physikal Layer"
    Label (195,285 195x20), "ASCII Frame"
    Frame (65,75 120x20)
        shows CtaSysConfig.visUDINT(visfbUDINTIn := fbModBusServerIn.scParameter.scSerial.fbudiBaudrate)
    Frame (65,40 120x20)
        shows CtaSysConfig.visBYTE(visfbBYTEIn := fbModBusServerIn.scParameter.scSerial.fbbyUnitId)
    Frame (165,5 20x20)
        shows CtaSysConfig.visBOOL(visfbBOOLIn := fbModBusServerIn.scParameter.scSerial.fbxEnable)
    Label (195,320 195x20), "Serial WatchDog"
    Label (195,355 195x20), "Serial WatchDog Time"
    Frame (5,355 180x20)
        shows CtaSysConfig.visTIME(visfbTIMEIn := fbModBusServerIn.scParameter.scTcp.fbtWatchDog)
    Frame (165,320 20x20)
        shows CtaSysConfig.visBOOL(visfbBOOLIn := fbModBusServerIn.scParameter.scTcp.fbxEnableWatchDog)
    Frame (165,285 20x20)
        shows CtaSysConfig.visBOOL(visfbBOOLIn := fbModBusServerIn.scParameter.scSerial.fbxRtuOrAscii)
    Frame (5,250 180x20), text list: 'txtPhysikalLayer', text index: fbModBusServerIn.scParameter.scSerial.fbiPhysikal.proValue
        shows CtaSysConfig.visENUMERATION(visfbENUIn := fbModBusServerIn.scParameter.scSerial.fbiPhysikal)
    Frame (5,215 180x20), text list: 'txtHandshake', text index: fbModBusServerIn.scParameter.scSerial.fbiHandshake.proValue
        shows CtaSysConfig.visENUMERATION(visfbENUIn := fbModBusServerIn.scParameter.scSerial.fbiHandshake)
    Frame (5,180 180x20), text list: 'txtStopBits', text index: fbModBusServerIn.scParameter.scSerial.fbiStopBits.proValue
        shows CtaSysConfig.visENUMERATION(visfbENUIn := fbModBusServerIn.scParameter.scSerial.fbiStopBits)
    Frame (5,145 180x20), text list: 'txtParity', text index: fbModBusServerIn.scParameter.scSerial.fbiParity.proValue
        shows CtaSysConfig.visENUMERATION(visfbENUIn := fbModBusServerIn.scParameter.scSerial.fbiParity)
    Frame (65,110 120x20)
        shows CtaSysConfig.visUSINT(visfbUSINTIn := fbModBusServerIn.scParameter.scSerial.fbusiDataBits)
END_VISUALIZATION

